// ---- DUTs/GreenMaster/IO/GreenMasterAI_Base.TcPOU
FUNCTION_BLOCK GreenMasterAI_Base
VAR_IN_OUT
	AIn: AnalogInputs;
END_VAR
VAR_INPUT
END_VAR
VAR_OUTPUT
	F_BT1_Error: BOOL;
	F_BT1: LREAL;
	T_BT2_Error: BOOL;
	T_BT2: LREAL;
	T_BT3_Error: BOOL;
	T_BT3: LREAL;
	H_BT1_Error: BOOL;
	H_BT1: LREAL;
	T_BT1_Error: BOOL;
	T_BT1: LREAL;
	BT1_Error: BOOL;
	BT1: LREAL;
	BT2_Error: BOOL;
	BT2: LREAL;
	F_BT2_Error: BOOL;
	F_BT2: LREAL;
END_VAR
VAR
END_VAR

END_FUNCTION_BLOCK

// ---- DUTs/GreenMaster/IO/GreenMasterAIU_Base.TcPOU
FUNCTION_BLOCK GreenMasterAIU_Base
VAR_INPUT
	EN: BOOL;
	T_BP2_Override: BOOL;
	T_BP2_OverrideValue: LREAL;
END_VAR
VAR_OUTPUT
	T_BF1_Error: BOOL;
	T_BF1: LREAL;
	F_BF1_Error: BOOL;
	F_BF1: LREAL;
	T_BP1_Error: BOOL;
	T_BP1: LREAL;
	F_BP1_Error: BOOL;
	F_BP1: LREAL;
	T_BP2_Error: BOOL;
	T_BP2: LREAL;
	F_BP2_Error: BOOL;
	F_BP2: LREAL;
	F_BP3_Error: BOOL;
	F_BP3: LREAL;
	T_CurrentPower: LREAL;
	F_CurrentPower: LREAL;
	T_CurrentSpeed: LREAL;
	F_CurrentSpeed: LREAL;
END_VAR
VAR
END_VAR

END_FUNCTION_BLOCK

// ---- DUTs/Parameters/IO/AnalogOutputParametersFB.TcPOU
FUNCTION_BLOCK AnalogOutputParametersFB
VAR_INPUT
END_VAR
VAR_OUTPUT
END_VAR
VAR
END_VAR

METHOD Update : BOOL
VAR_INPUT
	AO: REFERENCE TO GreenMasterAO_Base;
	Parameters: REFERENCE TO GreenMasterBaseParameters;
	AOut: AnalogOutputParameters;
END_VAR
VAR
	NotFire: BOOL;
END_VAR
NotFire := NOT Main.GreenMaster.FireAlarm();
AO.F_QN1 := ifc_lreal(Parameters.IO.AOutOverride.F_QN1_Override AND NotFire, Parameters.IO.AOutOverride.F_QN1_OverrideValue, AOut.F_QN1);
AO.T_GQ1 := ifc_lreal(Parameters.IO.AOutOverride.T_GQ1_Override AND NotFire, Parameters.IO.AOutOverride.T_GQ1_OverrideValue, AOut.T_GQ1);
AO.F_GQ1 := ifc_lreal(Parameters.IO.AOutOverride.F_GQ1_Override AND NotFire, Parameters.IO.AOutOverride.F_GQ1_OverrideValue, AOut.F_GQ1);
AO.C_QN1 := ifc_lreal(Parameters.IO.AOutOverride.C_QN1_Override AND NotFire, Parameters.IO.AOutOverride.C_QN1_OverrideValue, AOut.C_QN1);
AO.H_QN1 := ifc_lreal(Parameters.IO.AOutOverride.H_QN1_Override AND NotFire, Parameters.IO.AOutOverride.H_QN1_OverrideValue, AOut.H_QN1);
END_METHOD

END_FUNCTION_BLOCK

// ---- DUTs/GreenMaster/IO/GreenMasterAO_Base.TcPOU
FUNCTION_BLOCK GreenMasterAO_Base
VAR_IN_OUT
	AOut: AnalogOutputs;
END_VAR
VAR_INPUT
	F_QN1: LREAL;
	T_GQ1: LREAL;
	F_GQ1: LREAL;
	C_QN1: LREAL;
	H_QN1: LREAL;	
END_VAR
VAR_OUTPUT
END_VAR
VAR
END_VAR

METHOD SetOverrideF_GQ1 : BOOL
VAR_INPUT
	Override: BOOL;
	OverrideValue: LREAL;
	Parameters: REFERENCE TO GreenMasterBaseParameters;
END_VAR
END_METHOD

METHOD SetOverrideF_QN1 : BOOL
VAR_INPUT
	Override: BOOL;
	OverrideValue: LREAL;
	Parameters: REFERENCE TO GreenMasterBaseParameters;
END_VAR
END_METHOD

METHOD SetOverrideH_QN1 : BOOL
VAR_INPUT
	Override: BOOL;
	OverrideValue: LREAL;
	Parameters: REFERENCE TO GreenMasterBaseParameters;
END_VAR
END_METHOD

METHOD SetOverrideT_GQ1 : BOOL
VAR_INPUT
	Override: BOOL;
	OverrideValue: LREAL;
	Parameters: REFERENCE TO GreenMasterBaseParameters;
END_VAR
END_METHOD

END_FUNCTION_BLOCK

// ---- DUTs/Utilities/ifc_lreal.TcPOU
FUNCTION ifc_lreal : LREAL
VAR_INPUT
	Condition: BOOL;
	ValueTrue: LREAL;
	ValueFalse: LREAL;
END_VAR
VAR
END_VAR

IF Condition THEN
	ifc_lreal := ValueTrue;
ELSE
	ifc_lreal := ValueFalse;
END_IF

END_FUNCTION

// ---- DUTs/Utilities/BoolToErrorText.TcPOU
FUNCTION BoolToErrorText : STRING
VAR_INPUT
	Error: BOOL;
END_VAR
VAR
END_VAR

IF Error THEN
	BoolToErrorText := 'Error';
ELSE
	BoolToErrorText := 'OK';
END_IF

END_FUNCTION

// ---- DUTs/Parameters/Simulation/SimulationFB.TcPOU
FUNCTION_BLOCK SimulationFB
VAR_IN_OUT
	Parameters: GreenMasterBaseParameters;
END_VAR
VAR_INPUT
	Simulation: SimulationParameters;	
END_VAR
VAR_OUTPUT
END_VAR
VAR
END_VAR

Main.GreenMaster.Simulate(Parameters := Main.GreenMaster.GetParameters(),
	ParametersFB := Main.GreenMaster.GetParametersFB());

END_FUNCTION_BLOCK

// ---- DUTs/Parameters/SmokeControl/SmokeControlParametersBaseFB.TcPOU
FUNCTION_BLOCK SmokeControlParametersBaseFB
VAR_INPUT
END_VAR
VAR_OUTPUT
	NetLink: NetLinkParametersFB;
	DamperModules: SxDuoParametersFB;
END_VAR
VAR
END_VAR

END_FUNCTION_BLOCK

// ---- DUTs/Parameters/SmokeControl/NetLinkParametersFB.TcPOU
FUNCTION_BLOCK NetLinkParametersFB
VAR_INPUT
END_VAR
VAR_OUTPUT
END_VAR
VAR
END_VAR

METHOD Update : BOOL
VAR_INPUT
	Parameters: REFERENCE TO GreenMasterBaseParameters;
END_VAR
END_METHOD

END_FUNCTION_BLOCK

// ---- DUTs/Parameters/SmokeControl/SxDuoParametersFB.TcPOU
FUNCTION_BLOCK SxDuoParametersFB
VAR_INPUT
END_VAR
VAR_OUTPUT
	Unit01: SxDuoUnitFB;
	Unit02: SxDuoUnitFB;
	Unit03: SxDuoUnitFB;
	Unit04: SxDuoUnitFB;
	Unit05: SxDuoUnitFB;
	Unit06: SxDuoUnitFB;
	Unit07: SxDuoUnitFB;
	Unit08: SxDuoUnitFB;
	Unit09: SxDuoUnitFB;
	Unit10: SxDuoUnitFB;
	Unit11: SxDuoUnitFB;
	Unit12: SxDuoUnitFB;
	Unit13: SxDuoUnitFB;
	Unit14: SxDuoUnitFB;
	Unit15: SxDuoUnitFB;
END_VAR
VAR
END_VAR

END_FUNCTION_BLOCK

// ---- DUTs/Parameters/SmokeControl/SxDuoUnitFB.TcPOU
FUNCTION_BLOCK SxDuoUnitFB
VAR_INPUT
	Simulation: REFERENCE TO SimulationParameters;
END_VAR
VAR_OUTPUT
END_VAR
VAR
END_VAR

Simulation.ENO := Simulation.EN;

METHOD Update : BOOL
VAR_INPUT
	Parameters: REFERENCE TO GreenMasterBaseParameters;
	DamperModule: REFERENCE TO DamperModule;
	SxDuoUnit: REFERENCE TO SxDuoUnit;
END_VAR
SxDuoUnit.Error := DamperModule.Error;
SxDuoUnit.Fire := DamperModule.Fire;
SxDuoUnit.SxDuoStatus := DamperModule.SxDuoStatus;
DamperModule.SxDuoCommand := SxDuoUnit.SxDuoCommand;
SxDuoUnit.Text := DamperModule.Text;
SxDuoUnit.Text_CP1252 := DamperModule.Text_CP1252;
END_METHOD

END_FUNCTION_BLOCK

// ---- DUTs/Smoke Control/DamperModule.TcPOU
FUNCTION_BLOCK DamperModule
VAR_INPUT
	EN: BOOL;
	UnitID: BYTE;
	ModbusTCP: REFERENCE TO Modbus;
	Exercise: BOOL;
	ResetSmokeDetector: bool;
	SxDuoCommand: SxDuoCommand;
	{attribute 'TcEncoding':='UTF-8'}
	WriteText: STRING;
END_VAR
VAR_OUTPUT
	ENO: BOOL;
	Error: BOOL;
	Fire: BOOL;
	Exercising: BOOL;
	DamperError: BOOL;
	ServiceAlarm: BOOL;
	{attribute 'TcEncoding':='UTF-8'}
	Text: STRING;
	Text_CP1252: STRING;
	SxDuoStatus: SxDuoStatus;
END_VAR
VAR
	ModbusReadBits3: ModbusReadBits;
	ModbusWriteBits3: ModbusWriteBits;
	ModbusReadWordArray_0: ModbusReadWordArray;
END_VAR
VAR // added by the converter: edge detectors and wires of the graphical bodies
    _s1 : SxDuoStatus;
    _w1, _w2 : ANY;
END_VAR


// PAGE
ModbusWriteBits3(
    EN := EN,
    Modbus := ModbusTCP,
    UnitID := UnitID,
    Register := 44,
    b1 := ???,
    b2 := _w1,
    b4 := _w2); // ModbusWriteBits
ModbusReadBits3(EN := EN, Modbus := ModbusTCP, UnitID := UnitID, Register := 32); // ModbusReadBits
Error := ModbusReadBits3.Error;
Fire := ModbusReadBits3.b1;
_w2 := Exercise OR ???;
Exercising := ModbusReadBits3.b4;
DamperError := ModbusReadBits3.b6;
// compose _s1 : SxDuoStatus
_s1.FireAlarm := ModbusReadBits3.b1;
_s1.Damper1Alarm := ModbusReadBits3.b3;
_s1.Exercising := ModbusReadBits3.b4;
_s1.Damper2Alarm := ModbusReadBits3.b5;
_s1.Damper1Open := ModbusReadBits3.b9;
_s1.Damper1Closed := ModbusReadBits3.b8;
_s1.Damper2Open := ModbusReadBits3.b11;
_s1.Damper2Closed := ModbusReadBits3.b10;
_s1.ServiceAlarm := ModbusReadBits3.b14;
SxDuoStatus := _s1;
_w1 := ResetSmokeDetector OR ???;
ServiceAlarm := ModbusReadBits3.b14;
ModbusReadWordArray_0(
    EN := EN,
    Modbus := ModbusTCP,
    UnitID := UnitID,
    RegisterType := ModbusRegisterType.HoldingRegister,
    Register := 16#8000 + 16#110,
    ParameterCount := 16,
    UpdateInterval := LTIME#1m,
    WriteText := WriteText); // ModbusReadWordArray
Text := ModbusReadWordArray_0.Text;
Text_CP1252 := ModbusReadWordArray_0.Text_CP1252;

METHOD StartWrite : BOOL
VAR_INPUT
END_VAR
ModbusWriteBits3.EN := TRUE;
END_METHOD

END_FUNCTION_BLOCK

// ---- DUTs/ModbusTCP/ModbusTCP.TcPOU
FUNCTION_BLOCK ModbusTCP EXTENDS Modbus
VAR_INPUT
	EN: BOOL;
	{attribute 'TcEncoding':='UTF-8'}
	IP: STRING;
	Port: UINT := 502;
END_VAR
VAR_OUTPUT
	ENO: BOOL;
	Error: BOOL;
END_VAR
VAR
	ModbusMaster: FB_MBReadRegs;
	ModbusMasterWrite: FB_MBWriteRegs;
	{attribute 'TcEncoding':='UTF-8'}
	stMbErrId: STRING;
	aRegisterArray1: ARRAY [1..125] OF WORD;
	aRegisterCoil: ARRAY [1..250] OF BYTE;
	WaitModbusBusy: TON;
	cbRead: INT;
	Param: REFERENCE TO ModbusIo;
	State: INT;
	ReplyTON: LTON;
	LastReadCount: LINT;
END_VAR
VAR PERSISTENT
	tTimeBetweenReads: TIME := T#100MS;
END_VAR

SUPER^();
ENO := EN;
ReplyTON(IN := ReadCount = LastReadCount, PT := LTIME#20S, Q => Error);
LastReadCount := ReadCount;
WaitModbusBusy();
CASE State OF
	0:
		IF EN THEN		
			CurrentIoIndex := 0;
			IF IO[CurrentIoIndex] <> 0 THEN
				State := 5;
			END_IF	
		END_IF
	5:	(* Wait between reads *)
		WaitModbusBusy(IN := TRUE, PT := tTimeBetweenReads, Q=> , ET=> );	
		IF WaitModbusBusy.Q = TRUE THEN
			IF TIME_TO_LTIME(NowDT() - IO[CurrentIoIndex]^.LastUpdate) > IO[CurrentIoIndex]^.UpdateInterval THEN	
				IO[CurrentIoIndex]^.SetLastUpdate(NowDT());			
				IF NOT IO[CurrentIoIndex]^.Write THEN
					State := 10;
				ELSE
					State := 110;			
				END_IF
			ELSE
				State := 30;
			END_IF
			WaitModbusBusy(IN := FALSE);
		END_IF		
	
	10:
		Param REF= IO[CurrentIoIndex]^; 
		IF NOT Param.EN OR Param.UnitID = 0 THEN
			Param.ValueWord := 0;
			Param.ErrorOUT := FALSE;
			State := 30;
		ELSE
			ModbusMaster(
			sIPAddr:= IP, 
			nTCPPort:= 502, 
			nUnitID:= Param.UnitID, 
			nQuantity:= Param.ParameterCount, 
			nMBAddr:= Param.Register, 
			cbLength:= 2 * Param.ParameterCount, 
			pDestAddr:= ADR(aRegisterArray1), 
			bExecute:= TRUE, 
			tTimeout:= T#1000MS);
			IF  ModbusMaster.bBUSY THEN
				State := State + 10;
			END_IF
		END_IF
	20:
		ModbusMaster();
		IF ModbusMaster.bError THEN
			stMbErrId := concat('Error ', UDINT_TO_STRING(ModbusMaster.nErrId));
			ModbusMaster(bExecute := FALSE);
			Param.ValueWord := 0;
			Param.ErrorOUT := TRUE;
			ErrorCount := ErrorCount + 1;
			ModbusMaster.bExecute:= FALSE;
			State := 30;
		ELSIF NOT ModbusMaster.bBUSY THEN
			ModbusMaster(bExecute := FALSE);
			Param.ValueWord := aRegisterArray1[1];
			Param.ValueWordArray := aRegisterArray1;
			Param.ErrorOUT := FALSE;
			ReadCount := ReadCount + 1;
			ModbusMaster(bExecute:= FALSE);
			State := 30;
		END_IF
	30:
		CurrentIoIndex := CurrentIoIndex + 1;
		IF CurrentIoIndex >= IO_COUNT THEN
			CurrentIoIndex := 0;
		END_IF
		IF IO[CurrentIoIndex] <> 0 THEN
			State := 5;
		ELSE				
			State := 0;
		END_IF
	110:
		Param REF= IO[CurrentIoIndex]^; 
		IF NOT Param.EN OR Param.UnitID = 0 THEN
			Param.ValueWord := 0;
			Param.ErrorOUT := FALSE;
			State := 30;
		ELSE
			aRegisterArray1[1] := Param.ValueWord;
			ModbusMasterWrite(
			sIPAddr:= IP, 
			nTCPPort:= 502, 
			nUnitID:= Param.UnitID, 
			nQuantity:= Param.ParameterCount, 
			nMBAddr:= Param.Register, 
			cbLength:= 2 * Param.ParameterCount, 
			pSrcAddr:= ADR(aRegisterArray1), 
			bExecute:= TRUE, 
			tTimeout:= T#1000MS);
			IF  ModbusMasterWrite.bBUSY THEN
				State := State + 10;
			END_IF
		END_IF
	120:
		ModbusMasterWrite();
		IF ModbusMasterWrite.bError THEN
			stMbErrId := concat('Error ', UDINT_TO_STRING(ModbusMaster.nErrId));
			ModbusMasterWrite(bExecute := FALSE);
			Param.ValueWord := 0;
			Param.ErrorOUT := TRUE;
			ErrorCount := ErrorCount + 1;
			ModbusMasterWrite.bExecute:= FALSE;
			State := 30;
		ELSIF NOT ModbusMasterWrite.bBUSY THEN
			ModbusMasterWrite(bExecute := FALSE);
			Param.ValueWord := aRegisterArray1[1];
			Param.ValueWordArray := aRegisterArray1;
			Param.ErrorOUT := FALSE;
			ReadCount := ReadCount + 1;
			ModbusMasterWrite(bExecute:= FALSE);
			State := 30;
		END_IF
		Param.EN := FALSE;
		Param.Write := FALSE;
END_CASE

END_FUNCTION_BLOCK

// ---- DUTs/ModbusRTU/Modbus.TcPOU
FUNCTION_BLOCK Modbus
VAR_INPUT
END_VAR
VAR_OUTPUT
	ReadCount: LINT;
	ErrorCount: LINT;
END_VAR
VAR CONSTANT
	IO_COUNT: INT := 100;
END_VAR
VAR
	Self: REFERENCE TO Modbus;
	IO: ARRAY [0..IO_COUNT - 1] OF POINTER TO ModbusIo;
	IOIndex: INT;
	CurrentIoIndex: INT;
END_VAR

Self REF= THIS^;

METHOD AddIO : BOOL
VAR_INPUT
	Self: pointer TO ModbusIO {flag write};
END_VAR
IF IOIndex < IO_COUNT THEN
	IO[IOIndex] := Self;
	IOIndex := IOIndex + 1;
END_IF
END_METHOD

END_FUNCTION_BLOCK

// ---- DUTs/ModbusRTU/ModbusIo.TcPOU
FUNCTION_BLOCK ModbusIo
VAR_INPUT
	EN: BOOL := TRUE;
	Modbus: REFERENCE TO Modbus;
	UnitID: BYTE;
	RegisterType: ModbusRegisterType;
	Register: WORD;
	Write: BOOL := FALSE;
	ParameterCount: WORD := 1;
	UpdateInterval: LTIME := LTIME#2S;
END_VAR
VAR_OUTPUT
	ENO: BOOL;
	Error: BOOL;
	LastUpdate: DT;
END_VAR
VAR_IN_OUT
END_VAR
VAR
	Registered: BOOL;
	ErrorCount: INT;
END_VAR
VAR PERSISTENT
END_VAR

IF EN AND __ISVALIDREF(Modbus) THEN
	IF NOT Registered THEN
		Modbus.AddIO(THIS);
		Registered := TRUE;	
	END_IF
END_IF
ENO := EN and not Error;

PROPERTY ErrorOut : BOOL
GET
ErrorOut := Error;
END_GET
SET
Error := ErrorOut;
END_SET
END_PROPERTY

METHOD GetErrorCount : INT
VAR_INPUT
END_VAR
GetErrorCount := ErrorCount;
END_METHOD

METHOD IncErrorCount : BOOL
VAR_INPUT
END_VAR
IF ErrorCount < 10 THEN
	ErrorCount := ErrorCount + 1;
END_IF
END_METHOD

METHOD ResetErrorCount : BOOL
VAR_INPUT
END_VAR
ErrorCount := 0;
END_METHOD

METHOD SetLastUpdate : BOOL
VAR_INPUT
	CurrentTime: DT;
END_VAR
LastUpdate := CurrentTime;
END_METHOD

PROPERTY ValueBoolOut : BOOL
GET
END_GET
SET
END_SET
END_PROPERTY

PROPERTY ValueWord : WORD
GET
END_GET
SET
END_SET
END_PROPERTY

PROPERTY ValueWordArray : ARRAY [1..125] OF WORD
GET
END_GET
SET
END_SET
END_PROPERTY

END_FUNCTION_BLOCK

// ---- DUTs/ModbusRTU/ModbusReadBits.TcPOU
FUNCTION_BLOCK ModbusReadBits EXTENDS ModbusIo
VAR_INPUT
END_VAR
VAR_OUTPUT
	b0: BOOL;
	b1: BOOL;
	b2: BOOL;
	b3: BOOL;
	b4: BOOL;
	b5: BOOL;
	b6: BOOL;
	b7: BOOL;
	b8: BOOL;
	b9: BOOL;
	b10: BOOL;
	b11: BOOL;
	b12: BOOL;
	b13: BOOL;
	b14: BOOL;
	b15: BOOL;
END_VAR
VAR
END_VAR

SUPER^();

PROPERTY ValueWord : WORD
GET
ValueWord := 0;
IF b0 THEN
	ValueWord := ValueWord OR 16#0001;
END_IF
IF b1 THEN
	ValueWord := ValueWord OR 16#0002;
END_IF
IF b2 THEN
	ValueWord := ValueWord OR 16#0004;
END_IF
IF b3 THEN
	ValueWord := ValueWord OR 16#0008;
END_IF
IF b4 THEN
	ValueWord := ValueWord OR 16#0010;
END_IF
IF b5 THEN
	ValueWord := ValueWord OR 16#0020;
END_IF
IF b6 THEN
	ValueWord := ValueWord OR 16#0040;
END_IF
IF b7 THEN
	ValueWord := ValueWord OR 16#0080;
END_IF
IF b8 THEN
	ValueWord := ValueWord OR 16#0100;
END_IF
IF b9 THEN
	ValueWord := ValueWord OR 16#0200;
END_IF
IF b10 THEN
	ValueWord := ValueWord OR 16#0400;
END_IF
IF b11 THEN
	ValueWord := ValueWord OR 16#0800;
END_IF
IF b12 THEN
	ValueWord := ValueWord OR 16#1000;
END_IF
IF b13 THEN
	ValueWord := ValueWord OR 16#2000;
END_IF
IF b14 THEN
	ValueWord := ValueWord OR 16#4000;
END_IF
IF b15 THEN
	ValueWord := ValueWord OR 16#8000;
END_IF
END_GET
SET
b0 := (ValueWord AND 16#0001) <> 0;
b1 := (ValueWord AND 16#0002) <> 0;
b2 := (ValueWord AND 16#0004) <> 0;
b3 := (ValueWord AND 16#0008) <> 0;
b4 := (ValueWord AND 16#0010) <> 0;
b5 := (ValueWord AND 16#0020) <> 0;
b6 := (ValueWord AND 16#0040) <> 0;
b7 := (ValueWord AND 16#0080) <> 0;
b8 := (ValueWord AND 16#0100) <> 0;
b9 := (ValueWord AND 16#0200) <> 0;
b10 := (ValueWord AND 16#0400) <> 0;
b11 := (ValueWord AND 16#0800) <> 0;
b12 := (ValueWord AND 16#1000) <> 0;
b13 := (ValueWord AND 16#2000) <> 0;
b14 := (ValueWord AND 16#4000) <> 0;
b15 := (ValueWord AND 16#8000) <> 0;
END_SET
END_PROPERTY

END_FUNCTION_BLOCK

// ---- DUTs/ModbusRTU/ModbusWriteBits.TcPOU
FUNCTION_BLOCK ModbusWriteBits EXTENDS ModbusIo
VAR_INPUT
	b0: BOOL;
	b1: BOOL;
	b2: BOOL;
	b3: BOOL;
	b4: BOOL;
	b5: BOOL;
	b6: BOOL;
	b7: BOOL;
	b8: BOOL;
	b9: BOOL;
	b10: BOOL;
	b11: BOOL;
	b12: BOOL;
	b13: BOOL;
	b14: BOOL;
	b15: BOOL;
END_VAR
VAR_OUTPUT
END_VAR
VAR
	Pre_b0: BOOL;
	Pre_b1: BOOL;
	Pre_b2: BOOL;
	Pre_b3: BOOL;
	Pre_b4: BOOL;
	Pre_b5: BOOL;
	Pre_b6: BOOL;
	Pre_b7: BOOL;
	Pre_b8: BOOL;
	Pre_b9: BOOL;
	Pre_b10: BOOL;
	Pre_b11: BOOL;
	Pre_b12: BOOL;
	Pre_b13: BOOL;
	Pre_b14: BOOL;
	Pre_b15: BOOL;
END_VAR

SUPER^();
IF 
	(b0 <> Pre_b0) OR
	(b1 <> Pre_b1) OR
	(b2 <> Pre_b2) OR
	(b3 <> Pre_b3) OR
	(b4 <> Pre_b4) OR
	(b5 <> Pre_b5) OR
	(b6 <> Pre_b6) OR
	(b7 <> Pre_b7) OR
	(b8 <> Pre_b8) OR
	(b9 <> Pre_b9) OR
	(b10 <> Pre_b10) OR
	(b11 <> Pre_b11) OR
	(b12 <> Pre_b12) OR
	(b13 <> Pre_b13) OR
	(b14 <> Pre_b14) OR
	(b15 <> Pre_b15) THEN
	Pre_b0 := b0;
	Pre_b1 := b1;
	Pre_b2 := b2;
	Pre_b3 := b3;
	Pre_b4 := b4;
	Pre_b5 := b5;
	Pre_b6 := b6;
	Pre_b7 := b7;
	Pre_b8 := b8;
	Pre_b9 := b9;
	Pre_b10 := b10;
	Pre_b11 := b11;
	Pre_b12 := b12;
	Pre_b13 := b13;
	Pre_b14 := b14;
	Pre_b15 := b15;
	Write := TRUE;
END_IF

PROPERTY ValueWord : WORD
GET
ValueWord := 0;
IF b0 THEN
	ValueWord := ValueWord OR 16#0001;
END_IF
IF b1 THEN
	ValueWord := ValueWord OR 16#0002;
END_IF
IF b2 THEN
	ValueWord := ValueWord OR 16#0004;
END_IF
IF b3 THEN
	ValueWord := ValueWord OR 16#0008;
END_IF
IF b4 THEN
	ValueWord := ValueWord OR 16#0010;
END_IF
IF b5 THEN
	ValueWord := ValueWord OR 16#0020;
END_IF
IF b6 THEN
	ValueWord := ValueWord OR 16#0040;
END_IF
IF b7 THEN
	ValueWord := ValueWord OR 16#0080;
END_IF
IF b8 THEN
	ValueWord := ValueWord OR 16#0100;
END_IF
IF b9 THEN
	ValueWord := ValueWord OR 16#0200;
END_IF
IF b10 THEN
	ValueWord := ValueWord OR 16#0400;
END_IF
IF b11 THEN
	ValueWord := ValueWord OR 16#0800;
END_IF
IF b12 THEN
	ValueWord := ValueWord OR 16#1000;
END_IF
IF b13 THEN
	ValueWord := ValueWord OR 16#2000;
END_IF
IF b14 THEN
	ValueWord := ValueWord OR 16#4000;
END_IF
IF b15 THEN
	ValueWord := ValueWord OR 16#8000;
END_IF
END_GET
SET
b0 := (ValueWord AND 16#0001) <> 0;
b1 := (ValueWord AND 16#0002) <> 0;
b2 := (ValueWord AND 16#0004) <> 0;
b3 := (ValueWord AND 16#0008) <> 0;
b4 := (ValueWord AND 16#0010) <> 0;
b5 := (ValueWord AND 16#0020) <> 0;
b6 := (ValueWord AND 16#0040) <> 0;
b7 := (ValueWord AND 16#0080) <> 0;
b8 := (ValueWord AND 16#0100) <> 0;
b9 := (ValueWord AND 16#0200) <> 0;
b10 := (ValueWord AND 16#0400) <> 0;
b11 := (ValueWord AND 16#0800) <> 0;
b12 := (ValueWord AND 16#1000) <> 0;
b13 := (ValueWord AND 16#2000) <> 0;
b14 := (ValueWord AND 16#4000) <> 0;
b15 := (ValueWord AND 16#8000) <> 0;
END_SET
END_PROPERTY

END_FUNCTION_BLOCK

// ---- DUTs/ModbusRTU/ModbusReadWordArray.TcPOU
FUNCTION_BLOCK ModbusReadWordArray EXTENDS ModbusIo
VAR_INPUT
	{attribute 'TcEncoding':='UTF-8'}
	WriteText: STRING;
END_VAR
VAR_OUTPUT
	Value: ARRAY [1..125] OF WORD;
	{attribute 'TcEncoding':='UTF-8'}
	Text: STRING;
	Text_CP1252: STRING;
END_VAR
VAR
END_VAR
VAR PERSISTENT
END_VAR

SUPER^();
Text := GetText();
Text_CP1252 := GetText_CP1252();
SetText(WriteText);

{attribute 'TcEncoding':='UTF-8'}
METHOD GetText : string
VAR_INPUT
END_VAR
VAR
	//{attribute 'TcEncoding':='UTF-8'}
	Str: STRING;
	arr: ARRAY [1..125] OF WORD;
	p: POINTER TO ARRAY [0..MAX_STRING_LENGTH] OF BYTE;
	n: INT;
	{attribute 'TcEncoding':='UTF-8'}
	Utf8: STRING;
END_VAR
arr := Value;
FOR n := 1 TO 125 DO
	arr[n] := SHR(arr[n] AND 16#FF00, 8) + SHL(arr[n] AND 16#00FF, 8);
END_FOR
p := ADR(arr);
Str := BYTEARR_TO_MAXSTRING(p^);
STRING_TO_UTF8(ADR(Utf8), ADR(Str), SIZEOF(Utf8));
GetText := Utf8;
END_METHOD

METHOD GetText_CP1252 : STRING
VAR_INPUT
END_VAR
VAR
	Str: STRING;
	arr: ARRAY [1..125] OF WORD;
	p: POINTER TO ARRAY [0..MAX_STRING_LENGTH] OF BYTE;
	n: INT;
END_VAR
arr := Value;
FOR n := 1 TO 125 DO
	arr[n] := SHR(arr[n] AND 16#FF00, 8) + SHL(arr[n] AND 16#00FF, 8);
END_FOR
p := ADR(arr);
Str := BYTEARR_TO_MAXSTRING(p^);
GetText_CP1252 := Str;
END_METHOD

METHOD SetText : BOOL
VAR_INPUT
	{attribute 'TcEncoding':='UTF-8'}
	NewText: STRING;
END_VAR
VAR
	Str: STRING;
	TempValue, TestValue: ARRAY [1..125] OF WORD;
	bArr: ARRAY [0..MAX_STRING_LENGTH] OF BYTE;
	n: INT;
	{attribute 'TcEncoding':='UTF-8'}
	nDstLen: UDINT;
	byte0, byte1: BYTE;
	numWords: INT;
END_VAR
(*
IF UTF8_TO_STRING(ADR(Str), ADR(NewText), SIZEOF(Str), nDstLen => nDstLen) THEN	
	bArr := MAXSTRING_TO_BYTEARR(Str);
	bArr[nDstLen] := 0;
	nDstLen := nDstLen + 1;
	TempValue := Value;
	numWords := UDINT_TO_INT(nDstLen / 2);
	IF (nDstLen AND 1) <> 0 THEN
		numWords := numWords + 1;
	END_IF
	FOR n := 0 TO numWords - 1 DO
		IF (n * 2 + 1) < UDINT_TO_INT(nDstLen) THEN
			byte0 := bArr[n * 2 + 1];
		ELSE
			byte0 := 0;		
		END_IF
		byte1 := bArr[n * 2];
		TempValue[n + 1] := SHL(BYTE_TO_WORD(byte0), 8) + byte1;
	END_FOR
	IF NOT AnyEqual(TempValue, Value) THEN
		TestValue := TempValue;
		//Value := TempValue;
		//Write := TRUE;
	END_IF
END_IF
*)
END_METHOD

PROPERTY TextValue : STRING
GET
TextValue := GetText();
END_GET
SET
SetText(TextValue);
END_SET
END_PROPERTY

PROPERTY ValueWordArray : array [1..125] of WORD
GET
ValueWordArray := Value;
END_GET
SET
Value := ValueWordArray;
END_SET
END_PROPERTY

END_FUNCTION_BLOCK

// ---- DUTs/Utilities/WriteBoolIf.TcPOU
FUNCTION_BLOCK WriteBoolIf
VAR_IN_OUT
	Out: BOOL;
END_VAR
VAR_INPUT
	EN: BOOL := TRUE;
	In: BOOL;
END_VAR
VAR_OUTPUT
	ENO: BOOL;
END_VAR
VAR
END_VAR

ENO := EN;
IF EN THEN
	Out := In;
END_IF

END_FUNCTION_BLOCK

// ---- DUTs/Exercise/ExerciseF_P1.TcPOU
FUNCTION_BLOCK ExerciseF_P1
VAR_IN_OUT
	Parameters: GreenMasterBaseParameters;
END_VAR
VAR_INPUT
	EN: BOOL := TRUE;
	ForceExercise: BOOL;
END_VAR
VAR_OUTPUT
	Exercising: BOOL;
END_VAR
VAR
	ExerciseTimer: Timer;
	LocalTime: FB_LocalSystemTime;
	Elapsed: LINT;
	CurrentState: INT;
	StateTimer: TImer;
	DetectedDamperError: BOOL;
	FirstTime: BOOL := TRUE;
END_VAR

LocalTime(bEnable := TRUE);
ExerciseTimer(EN := EN);
Elapsed := ExerciseTimer.ElapsedTime();

StateTimer();
IF EN THEN
	CASE CurrentState OF
		0:
			IF EN AND LocalTime.bValid THEN
				IF ((Parameters.System.Exercise.CirculationPumps.Interval > 0) AND ((ExerciseTimer.ElapsedTime() > (Parameters.System.Exercise.CirculationPumps.Interval * 3600 * 1000)) OR FirstTime) AND 
					(
						(WORD_TO_INT(LocalTime.systemTime.wHour) = Parameters.System.Exercise.CirculationPumps.Hour) AND (WORD_TO_INT(LocalTime.systemTime.wMinute) = Parameters.System.Exercise.CirculationPumps.Minute)
					)) OR ForceExercise THEN
					FirstTime := FALSE;
					ForceExercise := FALSE;
					Exercising := TRUE;
					StateTimer.Restart();
					CurrentState := 1;
					Main.EventLog.LogEvent(EventTypes.Information, 'Exercising P1');
				END_IF			
			END_IF
		1:
			IF StateTimer.ElapsedTime() > 60 * 1000 THEN
				Exercising := FALSE;
				CurrentState := 0;
			END_IF
	END_CASE
END_IF

END_FUNCTION_BLOCK

// ---- DUTs/Events/EventLog.TcPOU
FUNCTION_BLOCK EventLog
VAR_IN_OUT
	EventLogData: EventLogData;	
END_VAR
VAR_INPUT
END_VAR
VAR_OUTPUT
END_VAR
VAR
	StartupDone: BOOL;
	EventLogDataRef: reference to EventLogData;	
	IncludeJSON: BOOL;
	sJSON: STRING(2000);
	fbJsonDataType: FB_JsonReadWriteDataType;
END_VAR

IF NOT StartupDone THEN
	EventLogDataRef REF= EventLogData;
	StartupDone := TRUE;
END_IF

METHOD LogEvent : BOOL
VAR_INPUT
	Kind: EventTypes := EventTypes.Information;
	Message: STRING;
END_VAR
VAR
	TempHead, TempTail: INT;
	n: uint;
END_VAR
IF __ISVALIDREF(EventLogDataRef) THEN
	TempTail := EventLogDataRef.Tail + 1;
	IF TempTail > Globals.EventsHigh THEN
		TempTail := Globals.EventsLow;
	END_IF
	
	IF TempTail = EventLogDataRef.Head THEN
		TempHead := EventLogDataRef.Head + 1;
		IF TempHead > Globals.EventsHigh THEN
			TempHead := Globals.EventsLow;
		END_IF
		EventLogDataRef.Head := TempHead;
	END_IF
	
	EventLogDataRef.Events[EventLogDataRef.Tail].Kind := Kind;
	EventLogDataRef.Events[EventLogDataRef.Tail].TimeStamp := NowDT();
	EventLogDataRef.Events[EventLogDataRef.Tail].Message := Message;
	n:= INT_TO_UINT(Len(sJSON));
	n :=  SIZEOF(EventLogDataRef.Events[EventLogDataRef.Tail].JSON);
	IF IncludeJSON AND (INT_TO_UINT(Len(sJSON)) < SIZEOF(Globals.EventLogStrings[EventLogDataRef.Tail])) THEN
		Globals.EventLogStrings[EventLogDataRef.Tail] := sJSON;
		EventLogDataRef.Events[EventLogDataRef.Tail].JSON := TRUE;
	ELSE
		EventLogDataRef.Events[EventLogDataRef.Tail].JSON := FALSE;
	END_IF
	
	EventLogDataRef.Tail := TempTail;
END_IF
END_METHOD

METHOD LogEventJSON : BOOL
VAR_INPUT
	Kind: EventTypes := EventTypes.Information;
	Message: STRING;
	VarType: STRING;
	VarSize: DWORD;
	VarAdr: POINTER TO DWORD;
END_VAR
VAR
	nLen: UDINT;
END_VAR
sJSON := '';
nLen := fbJsonDataType.CopyJsonStringFromSymbol(VarType, VarSize, VarAdr, sJSON,SIZEOF(sJSON));
IF nLen > 0 THEN
	IF sJSON[0] <> F_ToASC('{') THEN
		sJSON := concat(concat('{ "Value": ', sJSON), ' }');
	END_IF
END_IF
IncludeJSON := nLen > 0;
LogEvent(Kind := Kind, Message := Message);
IncludeJSON := FALSE;
END_METHOD

END_FUNCTION_BLOCK

// ---- DUTs/Utilities/DeviationMonitor.TcPOU
FUNCTION_BLOCK DeviationMonitor
VAR_INPUT
	EN: BOOL := TRUE;
	Value: LREAL;
	TargetValue: LREAL := 100;
	DiffAllowed: LREAL := 5;
	Mode: DeviationMonitorMode := DeviationMonitorMode.Diff;
	Hysteresis: LREAL := 2;
	OnDelay: LTIME := LTIME#10S;
	OffDelay: LTIME := LTIME#5S;
END_VAR
VAR_OUTPUT
	ENO: BOOL;
	Error: BOOL;
END_VAR
VAR
	TempError: BOOL;
	Hyst: Hysteresis;
	UseValue: LREAL;
	UseTargetValue: LREAL;
	OnTON: TON;
	OffTOF: TOF;
END_VAR

UseValue  := Value;
UseTargetValue := TargetValue;
IF Mode = DeviationMonitorMode.Diff THEN
	UseValue := ABS(UseValue - TargetValue);	
	UseTargetValue := DiffAllowed;
END_IF
Hyst(Value := UseValue, LimitValue := UseTargetValue, Offset := Hysteresis);
IF EN and (Main.GreenMaster.GetParameters().System.Operation.State = SystemStates.Run) THEN
	IF (Mode = DeviationMonitorMode.Above) OR (Mode = DeviationMonitorMode.Diff) THEN
		TempError := Hyst.Above;
	ELSIF Mode = DeviationMonitorMode.Below THEN
		TempError := Hyst.Below;	
	END_IF
	IF Main.GreenMaster.GetParameters().System.Operation.State <> SystemStates.Run THEN
		TempError := False;
	END_IF
	OnTON(IN := TempError, PT := TO_TIME(OnDelay));
	OffTOF(IN := NOT TempError, PT := TO_TIME(OnDelay));
	IF OnTON.Q THEN
		Error := TRUE;
	END_IF
	IF OffTOF.Q THEN
		Error := FALSE;
	END_IF
ELSE
	Error := FALSE;
END_IF
ENO := EN;

END_FUNCTION_BLOCK

// ---- DUTs/GreenMaster/IO/GreenMasterSmokeControl_Base.TcPOU
FUNCTION_BLOCK GreenMasterSmokeControl_Base
VAR_IN_OUT
	Parameters: GreenMasterBaseParameters;	
	ParametersSC: SmokeControlParametersBase;
END_VAR
VAR_INPUT
	EN: BOOL;
END_VAR
VAR_OUTPUT
	FireAlarm: BOOL;
END_VAR
VAR
END_VAR

END_FUNCTION_BLOCK

// ---- DUTs/Exercise/ExerciseF_QM2.TcPOU
FUNCTION_BLOCK ExerciseF_QM2
VAR_IN_OUT
	Parameters: GreenMasterBaseParameters;
END_VAR
VAR_INPUT
	EN: BOOL := TRUE;
	ForceExercise: BOOL;
END_VAR
VAR_OUTPUT
	Exercising: BOOL;
END_VAR
VAR
	ExerciseTimer: Timer;
	LocalTime: FB_LocalSystemTime;
	Elapsed: LINT;
	CurrentState: INT;
	StateTimer: TImer;
	DetectedDamperError: BOOL;
	FirstTime: BOOL := TRUE;
END_VAR

LocalTime(bEnable := TRUE);
ExerciseTimer(EN := EN);
Elapsed := ExerciseTimer.ElapsedTime();

StateTimer();
IF EN THEN
	CASE CurrentState OF
		0:
			IF EN AND LocalTime.bValid THEN
				IF ((Parameters.System.Exercise.FireBypassDamper.Interval > 0) AND ((ExerciseTimer.ElapsedTime() > (Parameters.System.Exercise.FireBypassDamper.Interval * 3600 * 1000)) OR FirstTime) AND 
					(
						(WORD_TO_INT(LocalTime.systemTime.wHour) = Parameters.System.Exercise.FireBypassDamper.Hour) AND (WORD_TO_INT(LocalTime.systemTime.wMinute) = Parameters.System.Exercise.FireBypassDamper.Minute)
					)) OR ForceExercise THEN
					FirstTime := FALSE;
					ForceExercise := FALSE;
					Exercising := TRUE;
					StateTimer.Restart();
					CurrentState := 1;
					Main.EventLog.LogEvent(EventTypes.Information, 'Exercising F_QM2');
				END_IF			
			END_IF
		1:
			IF StateTimer.ElapsedTime() > 10 * 1000 THEN
				ExerciseTimer.Restart();
				Parameters.IO.DOut.F_QM2 := FALSE;
				CurrentState := 2;
			END_IF
		2:
			IF StateTimer.ElapsedTime() > 30 * 1000 THEN
				CurrentState := 3;
			END_IF
		3:
			IF (StateTimer.ElapsedTime() > 180 * 1000) or Parameters.IO.DIn.F_QM2_Closed THEN
				Parameters.IO.DOut.F_QM2 := TRUE;
				Exercising := FALSE;
				CurrentState := 0;
			END_IF
	END_CASE
END_IF

END_FUNCTION_BLOCK

// ---- DUTs/Alarms/AlarmMonitor.TcPOU
FUNCTION_BLOCK AlarmMonitor
VAR_IN_OUT
	AlarmLog: AlarmLog;
	Parameters: GreenMasterBaseParameters;
END_VAR
VAR_INPUT
	EN: BOOL;
	Reset: BOOL;
END_VAR
VAR_OUTPUT
	ENO: BOOL;
	AlarmA: BOOL;
	AlarmB: BOOL;
	AlarmC: BOOL;
	AlarmD: BOOL;
END_VAR
VAR
	AlarmSignals1: REFERENCE TO AlarmSignals;
	StartupDone: BOOL;
	AlarmLogRef: REFERENCE TO AlarmLog;
	NoAlarms, Current: AlarmEvent;
	n: UINT;
	aTON: ARRAY [0..19] OF TON;
	bTON: ARRAY [0..11] OF TON;
	cTON: ARRAY [0..3] OF TON;
	CurrentDT, LastDT: DATE_AND_TIME;
	IncludeJSON: BOOL;
	sJSON: STRING(2000);
	fbJsonDataType: FB_JsonReadWriteDataType;
	StartTime: Timer;
	Latched, Last: AlarmEvent;
	LastIoStatus: IoStatus;
	
	AlarmCount: UINT := SIZEOF(AlarmSignals);
	LatchedStatusP: POINTER TO ARRAY [0..SIZEOF(AlarmSignals) - 1] OF BOOL;
	LatchedSignalP: POINTER TO ARRAY [0..SIZEOF(AlarmSignals) - 1] OF BOOL;
	StatusP: POINTER TO ARRAY [0..SIZEOF(AlarmSignals) - 1] OF BOOL;
	AutoResetP: POINTER TO ARRAY [0..SIZEOF(AlarmSignals) - 1] OF BOOL;
	EnabledP: POINTER TO ARRAY [0..SIZEOF(AlarmSignals) - 1] OF BOOL;
	CurrentP: POINTER TO ARRAY [0..SIZEOF(AlarmSignals) - 1] OF BOOL;
	PolarityP: POINTER TO ARRAY [0..SIZEOF(AlarmSignals) - 1] OF BOOL;
	DelayP: POINTER TO ARRAY [0..SIZEOF(AlarmSignals) - 1] OF TIME;
	TONs: ARRAY [0..SIZEOF(AlarmSignals) - 1] OF TON;
	StartupDelay: TON;
END_VAR

IF NOT StartupDone THEN
	AlarmLogRef REF= AlarmLog;
	StartupDone := TRUE;
	AlarmSignals1 REF= Parameters.Alarm.Status;
END_IF
StartupDelay(IN := TRUE, PT := T#5S);
IF StartupDelay.Q THEN
	LatchedStatusP := ADR(Latched.Status);
	DelayP := ADR(Parameters.Alarm.Delay);
	StatusP := ADR(Parameters.Alarm.Status);
	PolarityP := ADR(Parameters.Alarm.Polarity);
	CurrentP := ADR(Current.Signals);
	EnabledP := ADR(Parameters.Alarm.Enabled);
	FOR N := 0 TO AlarmCount - 1 DO
		LatchedStatusP^[n] := (StatusP^[n] <> PolarityP^[n]) AND EnabledP^[n];		
		TONs[n](IN := LatchedStatusP^[n], PT := DelayP^[n], Q => CurrentP^[n]);
	END_FOR
	
	IF (Parameters.IO.DIn.ResetAlarm OR Parameters.Alarm.Control.ResetAlarms) AND (AlarmA OR AlarmB OR AlarmC) THEN
		IF Parameters.IO.DIn.ResetAlarm THEN
			Main.EventLog.LogEvent(Message := 'Reset alarm via DI', Kind := EventTypes.Information);
		ELSE			
			Main.EventLog.LogEvent(Message := 'Reset alarm via web', Kind := EventTypes.Information);
		END_IF

		FOR N := 0 TO AlarmCount - 1 DO
			TONs[n](IN := FALSE);
		END_FOR
		Latched := NoAlarms;
		Parameters.Alarm.Control.ResetAlarms := FALSE;
		Globals.ResetAlarmsCounter := Globals.ResetAlarmsCounter + 1;
	END_IF
	
	// Transfer from Alarms to Latched according to autoreset and polarity definitions
	LatchedSignalP := ADR(Latched.Signals);
	AutoResetP := ADR(Parameters.Alarm.AutoReset);
	FOR N := 0 TO AlarmCount - 1 DO
		LatchedSignalP^[n] := LatchedSignalP^[n] AND NOT AutoResetP^[n] OR CurrentP^[n];
	END_FOR
	
	// Set parameters alarms
	Parameters.Alarm.Active.A := Latched.Signals.A;
	Parameters.Alarm.Active.B := Latched.Signals.B;
	Parameters.Alarm.Active.C := Latched.Signals.C;
	
	// Set alarms
	AlarmA := NOT AnyEqual(Latched.Signals.A, NoAlarms.Signals.A);
	AlarmB := NOT AnyEqual(Latched.Signals.B, NoAlarms.Signals.B);
	AlarmC := NOT AnyEqual(Latched.Signals.C, NoAlarms.Signals.C);
	AlarmD := FALSE;
	
	CurrentDT := NowDT();
	StartTime();
	IF (CurrentDT <> LastDT) AND (StartTime.ET > LTIME#20S) THEN
		// Add any alarm events to alarm log
		IF (NOT AnyEqual(Latched.Signals, Last.Signals)) or (NOT AnyEqual(Latched.Status, Last.Status)) THEN
			IF NOT Latched.Signals.C.SensorFailure THEN
				LogAlarm(Latched);
			ELSE
				LogAlarmJSON(Item := Latched, VarAdr := ADR(Parameters.IO.Status), VarSize := SIZEOF(Parameters.IO.Status), VarType := 'IoStatus');
			END_IF
			Last := Latched;
		END_IF
		LastDT := CurrentDT;
	END_IF
END_IF

METHOD LogAlarm : BOOL
VAR_INPUT
	Item: AlarmEvent;
END_VAR
VAR
	TempHead, TempTail: INT;
END_VAR
IF __ISVALIDREF(AlarmLogRef) THEN
	TempTail := AlarmLogRef.Tail + 1;
	IF TempTail > Globals.AlarmsHigh THEN
		TempTail := Globals.AlarmsLow;
	END_IF
	
	IF TempTail = AlarmLogRef.Head THEN
		TempHead := AlarmLogRef.Head + 1;
		IF TempHead > Globals.AlarmsHigh THEN
			TempHead := Globals.AlarmsLow;
		END_IF
		AlarmLogRef.Head := TempHead;
	END_IF
	Item.TimeStamp := NowDT();	
	AlarmLogRef.Alarms[AlarmLogRef.Tail] := Item;
	IF IncludeJSON AND (INT_TO_UINT(Len(sJSON)) < SIZEOF(Globals.AlarmLogStrings[AlarmLogRef.Tail]) ) THEN
		Globals.AlarmLogStrings[AlarmLogRef.Tail] := sJSON;
		AlarmLogRef.Alarms[AlarmLogRef.Tail].JSON := TRUE;
	ELSE
		AlarmLogRef.Alarms[AlarmLogRef.Tail].JSON := FALSE;
	END_IF
	
	AlarmLogRef.Tail := TempTail;
	Main.EventLog.LogEventJSON(Message := 'Alarm status changed', Kind := EventTypes.Error, VarAdr := ADR(Item.Signals), VarSize := SIZEOF(Item.Signals), VarType := 'AlarmSignals');
END_IF
END_METHOD

METHOD LogAlarmJSON : BOOL
VAR_INPUT
	Item: AlarmEvent;
	VarType: STRING;
	VarSize: DWORD;
	VarAdr: POINTER TO DWORD;
END_VAR
VAR
	nLen: UDINT;
END_VAR
sJSON := '';
nLen := fbJsonDataType.CopyJsonStringFromSymbol(VarType, VarSize, VarAdr, sJSON,SIZEOF(sJSON));
IncludeJSON := nLen > 0;
LogAlarm(Item := Item);
IncludeJSON := FALSE;
END_METHOD

END_FUNCTION_BLOCK

// ---- DUTs/System/AnyEqual.TcPOU
FUNCTION AnyEqual : BOOL
VAR_INPUT
	A: ANY;
	B: any;
END_VAR
VAR
	bDataTypesEquals: BOOL;
	bDataSizeEquals: BOOL;
	nCount: DINT;
	bDataContentEquals: BOOL;
END_VAR

IF A.TypeClass = B.TypeClass THEN
    bDataTypesEquals := TRUE;
END_IF
IF bDataTypesEquals THEN
    IF (A.diSize = B.diSize) THEN
        bDataSizeEquals := TRUE;
    END_IF
END_IF
IF bDataTypesEquals AND bDataSizeEquals THEN
    // Compare each byte in the ANY-types
	bDataContentEquals := TRUE;
    FOR nCount := 0 TO A.diSize-1 BY 1 DO
        IF A.pValue[nCount] <> B.pValue[nCount] THEN
            bDataContentEquals := FALSE;
            EXIT;
        END_IF
    END_FOR
END_IF
AnyEqual := bDataContentEquals AND bDataSizeEquals AND bDataTypesEquals;

END_FUNCTION

// ---- DUTs/Utilities/Scale.TcPOU
FUNCTION_BLOCK Scale
VAR_INPUT
	EN: BOOL := TRUE;
	x: LREAL;
	x1: LREAL;
	x2: LREAL;
	u1: LREAL;
	u2: LREAL;
END_VAR
VAR_OUTPUT
	ENO: bool;
	u: LREAL;
END_VAR
VAR
END_VAR

IF EN THEN
	IF u1 <= u2 THEN
		u := LimitValue((((x - x1) * (u2 - u1)) / (x2 - x1)) + u1, u1, u2);
	ELSE
		u := LimitValue(u1 - (((x - x1) * (u1 - u2)) / (x2 - x1)), u2, u1);
	END_IF
ELSE
	u := 0;
END_IF
ENO := EN;

END_FUNCTION_BLOCK

// ---- DUTs/Controllers/PidController.TcPOU
FUNCTION_BLOCK PidController
VAR_INPUT
	Param: ControllerParameters;
	EN: BOOL := TRUE;
	SP: LREAL;
	PV: LREAL;
	P: LREAL := 1;
	I: TIME := T#1M;
	Dtime: UDINT;
	DampingTime: TIME;
	SyncCV: LREAL;
	Sync: BOOL;
	Hold: BOOL;
	MinSpeed: LREAL := 0;
	MaxSpeed: LREAL := 1;
END_VAR
VAR_OUTPUT
	CV: LREAL;
	ENO: BOOL;
	Error: LREAL;
END_VAR
VAR
	Ctrl: FB_BA_PIDCtrl;
	TempCV: REAL;
END_VAR

Ctrl(	bEn := EN, 
		rW := LREAL_TO_REAL(SP), 
		rX := LREAL_TO_REAL(PV), 
		rKp := LREAL_TO_REAL(P), 
		udiTn_ms := TIME_TO_UDINT(I), 
		udiTv_ms := Dtime, 
		udiTd_ms := TIME_TO_UDINT(DampingTime), 
		rYMax := TO_REAL(MaxSpeed * 1000), 
		rYMin := TO_REAL(MinSpeed * 1000), 
		rSync := LREAL_TO_REAL(SyncCV * 1000), 
		bSync := Sync, 		
		rY => TempCV, 
		rE => Error
);
CV := TempCV / 1000;
ENO := EN;

END_FUNCTION_BLOCK

// ---- DUTs/Utilities/Average.TcPOU
FUNCTION_BLOCK Average
VAR_INPUT
	NewSample: LREAL;
END_VAR
VAR_OUTPUT
	Value: LREAL;
END_VAR
VAR
	Acc: lreal;
	LastSec: LINT;
END_VAR

IF LastSec = 0 THEN
	Acc := NewSample;
END_IF
IF Globals.SecondsCounter <> LastSec THEN
	Acc := Acc * 0.9;
	Acc := Acc + NewSample;
	Value := Acc / 10;
	LastSec := Globals.SecondsCounter;
END_IF

END_FUNCTION_BLOCK

// ---- DUTs/Utilities/WriteLRealOnlyIf.TcPOU
FUNCTION_BLOCK WriteLRealOnlyIf
VAR_IN_OUT
	Out: LREAL;	
END_VAR
VAR_INPUT
	EN: BOOL := TRUE;
	Value: LREAL;
END_VAR
VAR_OUTPUT
	ENO: bool;
END_VAR
VAR
END_VAR

ENO := EN;
IF EN THEN
	Out := Value;
END_IF

END_FUNCTION_BLOCK

// ---- POUs/SmokeControl.TcPOU
PROGRAM SmokeControl
VAR
	StartupDone: BOOL;
	GreenMasterSmokeControl: GreenMasterSmokeControl; 
	Parameters: REFERENCE TO GreenMasterBaseParameters;
	ParametersFB: REFERENCE TO GreenMasterBaseParametersFB;
	ParametersSC: REFERENCE TO SmokeControlParametersBase;
	ParametersSCFB: REFERENCE TO SmokeControlParametersBaseFB;
	ExerciseTimer: Timer;
	EN: BOOL;
	LocalTime: FB_LocalSystemTime;
	Elapsed: LINT;
	ForceExercise: BOOL;
	Exercising: BOOL;
	CurrentState: INT;
	StateTimer: TImer;
	DetectedDamperError: BOOL;
	DetectedDamperFireAlarm: BOOL;
END_VAR

IF NOT StartupDone THEN
	Parameters REF= Main.GreenMaster.GetParameters();
	ParametersSC REF= Main.GreenMaster.GetParametersSC();
	ParametersFB REF= Main.GreenMaster.GetParametersFB();
	ParametersSCFB REF= Main.GreenMaster.GetParametersSCFB();
	StartupDone := TRUE;
END_IF
EN := GetComponent(Name := ComponentNames.GM_SMOKE_CONTROL).EN;
LocalTime(bEnable := TRUE);
ExerciseTimer(EN := EN);
Elapsed := ExerciseTimer.ElapsedTime();
IF EN AND LocalTime.bValid THEN
	GreenMasterSmokeControl(EN := TRUE, Parameters := Parameters, ParametersSC := ParametersSC);
	GreenMasterSmokeControl.Update(Parameters, ParametersSC, ParametersFB, ParametersSCFB);
END_IF

IF GreenMasterSmokeControl.DamperError AND Parameters.Alarm.Active.B.DamperError THEN
	DetectedDamperError := TRUE;
END_IF
IF DetectedDamperError AND NOT Parameters.Alarm.Active.B.DamperError THEN
	DetectedDamperError := FALSE;
	ForceExercise := TRUE;
END_IF

IF GreenMasterSmokeControl.FireAlarm AND Parameters.Alarm.Active.A.FireLocal THEN
	DetectedDamperFireAlarm := TRUE;
END_IF
IF DetectedDamperFireAlarm AND NOT Parameters.Alarm.Active.A.FireLocal THEN
	DetectedDamperFireAlarm := FALSE;
	GreenMasterSmokeControl.ResetSmokeDetectors := TRUE;
	ForceExercise := TRUE;
END_IF
IF NOT Parameters.Alarm.Status.A.FireLocal THEN
	GreenMasterSmokeControl.ResetSmokeDetectors := FALSE;
END_IF

StateTimer();
CASE CurrentState OF
	0:
		IF EN AND LocalTime.bValid THEN
			IF ((ParametersSC.NetLink.Exercise.Interval > 0) AND (ExerciseTimer.ElapsedTime() > (ParametersSC.NetLink.Exercise.Interval * 3600 * 1000)) AND 
				(
					(WORD_TO_INT(LocalTime.systemTime.wHour) = ParametersSC.NetLink.Exercise.Hour) AND (WORD_TO_INT(LocalTime.systemTime.wMinute) = ParametersSC.NetLink.Exercise.Minute)
				)) OR ForceExercise THEN
				ForceExercise := FALSE;
				Exercising := TRUE;
				StateTimer.Restart();
				CurrentState := 1;
				Main.EventLog.LogEvent(EventTypes.Information, 'Exercising Smoke Control dampers');
			END_IF			
		END_IF
	1:
		IF StateTimer.ElapsedTime() > 10 * 1000 THEN
			GreenMasterSmokeControl.Exercise := TRUE;
			GreenMasterSmokeControl.Write();
			ExerciseTimer.Restart();
			CurrentState := 2;
		END_IF
	2:
		IF StateTimer.ElapsedTime() > 30 * 1000 THEN
			CurrentState := 3;
		END_IF
	3:
		IF (NOT GreenMasterSmokeControl.Exercising) OR (StateTimer.ElapsedTime() > 180 * 1000) THEN
			GreenMasterSmokeControl.Exercise := FALSE;
			Exercising := FALSE;
			CurrentState := 0;
		END_IF
END_CASE

END_PROGRAM

// ---- DUTs/GreenMaster/IO/GreenMasterSmokeControl.TcPOU
FUNCTION_BLOCK GreenMasterSmokeControl extends GreenMasterSmokeControl_Base
VAR_INPUT
	Exercise: BOOL;
	ResetSmokeDetectors: bool;
END_VAR
VAR_OUTPUT
	Exercising: BOOL;
	DamperError: BOOL;
	ServiceAlarm: BOOL;
END_VAR
VAR
	ModbusTCP: ModbusTCP;
	DamperControl: DamperControl;
	DamperModule_0: DamperModule;
	DamperModule_1: DamperModule;
	DamperModule_2: DamperModule;
	DamperModule_3: DamperModule;
	DamperModule_4: DamperModule;
	DamperModule_5: DamperModule;
	DamperModule_6: DamperModule;
	DamperModule_7: DamperModule;
	DamperModule_8: DamperModule;
	DamperModule_9: DamperModule;
	DamperModule_10: DamperModule;
	DamperModule_11: DamperModule;
	DamperModule_12: DamperModule;
	DamperModule_13: DamperModule;
	DamperModule_14: DamperModule;
END_VAR
VAR // added by the converter: edge detectors and wires of the graphical bodies
    _w1, _w2, _w3, _w4 : ANY;
END_VAR


// PAGE Modbus TCP
ModbusTCP(EN := EN, IP := ParametersSC.NetLink.ModbusTCP_IP);
Main.GreenMaster.GetParametersSC().NetLink.Error := ModbusTCP.Error;

// PAGE Smoke Detection
_w1 := DamperModule_0.DamperError OR DamperModule_1.DamperError OR DamperModule_2.DamperError OR DamperModule_3.DamperError OR DamperModule_4.DamperError OR DamperModule_5.DamperError OR DamperModule_6.DamperError OR DamperModule_7.DamperError OR DamperModule_8.DamperError OR DamperModule_9.DamperError OR DamperModule_10.DamperError OR DamperModule_11.DamperError OR DamperModule_12.DamperError OR DamperModule_13.DamperError OR DamperModule_14.DamperError;
DamperModule_4(
    EN := ParametersSC.DamperModules.Unit05.EN,
    UnitID := ParametersSC.DamperModules.Unit05.UnitID,
    ModbusTCP := ModbusTCP,
    Exercise := Exercise,
    ResetSmokeDetector := ResetSmokeDetectors,
    WriteText := ParametersSC.DamperModules.Unit05.Text); // DamperModule
_w2 := DamperModule_0.ServiceAlarm OR DamperModule_1.ServiceAlarm OR DamperModule_2.ServiceAlarm OR DamperModule_3.ServiceAlarm OR DamperModule_4.ServiceAlarm OR DamperModule_5.ServiceAlarm OR DamperModule_6.ServiceAlarm OR DamperModule_7.ServiceAlarm OR DamperModule_8.ServiceAlarm OR DamperModule_9.ServiceAlarm OR DamperModule_10.ServiceAlarm OR DamperModule_11.ServiceAlarm OR DamperModule_12.ServiceAlarm OR DamperModule_13.ServiceAlarm OR DamperModule_14.ServiceAlarm;
DamperModule_5(
    EN := ParametersSC.DamperModules.Unit06.EN,
    UnitID := ParametersSC.DamperModules.Unit06.UnitID,
    ModbusTCP := ModbusTCP,
    Exercise := Exercise,
    ResetSmokeDetector := ResetSmokeDetectors,
    WriteText := ParametersSC.DamperModules.Unit06.Text); // DamperModule
_w3 := DamperModule_0.Exercising OR DamperModule_1.Exercising OR DamperModule_2.Exercising OR DamperModule_3.Exercising OR DamperModule_4.Exercising OR DamperModule_5.Exercising OR DamperModule_6.Exercising OR DamperModule_7.Exercising OR DamperModule_8.Exercising OR DamperModule_9.Exercising OR DamperModule_10.Exercising OR DamperModule_11.Exercising OR DamperModule_12.Fire OR DamperModule_13.Fire OR DamperModule_14.Exercising;
DamperControl(EN := true);
FireAlarm := _w4;
_w4 := DamperModule_0.Fire OR DamperModule_1.Fire OR DamperModule_2.Fire OR DamperModule_3.Fire OR DamperModule_4.Fire OR DamperModule_5.Fire OR DamperModule_6.Fire OR DamperModule_7.Fire OR DamperModule_8.Fire OR DamperModule_9.Fire OR DamperModule_10.Fire OR DamperModule_11.Fire OR DamperModule_12.Fire OR DamperModule_13.Fire OR DamperModule_14.Fire;
Exercising := _w3;
DamperModule_6(
    EN := ParametersSC.DamperModules.Unit07.EN,
    UnitID := ParametersSC.DamperModules.Unit07.UnitID,
    ModbusTCP := ModbusTCP,
    Exercise := Exercise,
    ResetSmokeDetector := ResetSmokeDetectors,
    WriteText := ParametersSC.DamperModules.Unit07.Text); // DamperModule
DamperModule_7(
    EN := ParametersSC.DamperModules.Unit08.EN,
    UnitID := ParametersSC.DamperModules.Unit08.UnitID,
    ModbusTCP := ModbusTCP,
    Exercise := Exercise,
    ResetSmokeDetector := ResetSmokeDetectors,
    WriteText := ParametersSC.DamperModules.Unit08.Text); // DamperModule
DamperModule_8(
    EN := ParametersSC.DamperModules.Unit09.EN,
    UnitID := ParametersSC.DamperModules.Unit09.UnitID,
    ModbusTCP := ModbusTCP,
    Exercise := Exercise,
    ResetSmokeDetector := ResetSmokeDetectors,
    WriteText := ParametersSC.DamperModules.Unit09.Text); // DamperModule
DamperModule_13(
    EN := ParametersSC.DamperModules.Unit14.EN,
    UnitID := ParametersSC.DamperModules.Unit14.UnitID,
    ModbusTCP := ModbusTCP,
    Exercise := Exercise,
    ResetSmokeDetector := ResetSmokeDetectors,
    WriteText := ParametersSC.DamperModules.Unit14.Text); // DamperModule
DamperModule_14(
    EN := ParametersSC.DamperModules.Unit15.EN,
    UnitID := ParametersSC.DamperModules.Unit15.UnitID,
    ModbusTCP := ModbusTCP,
    Exercise := Exercise,
    ResetSmokeDetector := ResetSmokeDetectors,
    WriteText := ParametersSC.DamperModules.Unit15.Text); // DamperModule
DamperModule_11(
    EN := ParametersSC.DamperModules.Unit12.EN,
    UnitID := ParametersSC.DamperModules.Unit12.UnitID,
    ModbusTCP := ModbusTCP,
    Exercise := Exercise,
    ResetSmokeDetector := ResetSmokeDetectors,
    WriteText := ParametersSC.DamperModules.Unit12.Text); // DamperModule
DamperModule_12(
    EN := ParametersSC.DamperModules.Unit13.EN,
    UnitID := ParametersSC.DamperModules.Unit13.UnitID,
    ModbusTCP := ModbusTCP,
    Exercise := Exercise,
    ResetSmokeDetector := ResetSmokeDetectors,
    WriteText := ParametersSC.DamperModules.Unit13.Text); // DamperModule
DamperModule_9(
    EN := ParametersSC.DamperModules.Unit10.EN,
    UnitID := ParametersSC.DamperModules.Unit10.UnitID,
    ModbusTCP := ModbusTCP,
    Exercise := Exercise,
    ResetSmokeDetector := ResetSmokeDetectors,
    WriteText := ParametersSC.DamperModules.Unit10.Text); // DamperModule
DamperModule_10(
    EN := ParametersSC.DamperModules.Unit11.EN,
    UnitID := ParametersSC.DamperModules.Unit11.UnitID,
    ModbusTCP := ModbusTCP,
    Exercise := Exercise,
    ResetSmokeDetector := ResetSmokeDetectors,
    WriteText := ParametersSC.DamperModules.Unit11.Text); // DamperModule
ServiceAlarm := _w2;
DamperModule_2(
    EN := ParametersSC.DamperModules.Unit03.EN,
    UnitID := ParametersSC.DamperModules.Unit03.UnitID,
    ModbusTCP := ModbusTCP,
    Exercise := Exercise,
    ResetSmokeDetector := ResetSmokeDetectors,
    WriteText := ParametersSC.DamperModules.Unit03.Text); // DamperModule
DamperModule_3(
    EN := ParametersSC.DamperModules.Unit04.EN,
    UnitID := ParametersSC.DamperModules.Unit04.UnitID,
    ModbusTCP := ModbusTCP,
    Exercise := Exercise,
    ResetSmokeDetector := ResetSmokeDetectors,
    WriteText := ParametersSC.DamperModules.Unit04.Text); // DamperModule
DamperModule_0(
    EN := ParametersSC.DamperModules.Unit01.EN,
    UnitID := ParametersSC.DamperModules.Unit01.UnitID,
    ModbusTCP := ModbusTCP,
    Exercise := Exercise,
    ResetSmokeDetector := ResetSmokeDetectors,
    WriteText := ParametersSC.DamperModules.Unit01.Text); // DamperModule
DamperModule_1(
    EN := ParametersSC.DamperModules.Unit02.EN,
    UnitID := ParametersSC.DamperModules.Unit02.UnitID,
    ModbusTCP := ModbusTCP,
    Exercise := Exercise,
    ResetSmokeDetector := ResetSmokeDetectors,
    WriteText := ParametersSC.DamperModules.Unit02.Text); // DamperModule
DamperError := _w1;

METHOD Update : BOOL
VAR_INPUT
	Parameters: REFERENCE TO GreenMasterBaseParameters;
	ParametersSC: REFERENCE TO SmokeControlParametersBase;
	ParametersFB: REFERENCE TO GreenMasterBaseParametersFB;
	ParametersSCFB: REFERENCE TO SmokeControlParametersBaseFB;
END_VAR
VAR
	TempAlarm: bool;
END_VAR
ParametersSCFB.NetLink.Update(Parameters);
ParametersSCFB.DamperModules.Unit01.Update(Parameters, DamperModule_0, ParametersSC.DamperModules.Unit01);
ParametersSCFB.DamperModules.Unit02.Update(Parameters, DamperModule_1, ParametersSC.DamperModules.Unit02);
ParametersSCFB.DamperModules.Unit03.Update(Parameters, DamperModule_2, ParametersSC.DamperModules.Unit03);
ParametersSCFB.DamperModules.Unit04.Update(Parameters, DamperModule_3, ParametersSC.DamperModules.Unit04);
ParametersSCFB.DamperModules.Unit05.Update(Parameters, DamperModule_4, ParametersSC.DamperModules.Unit05);
ParametersSCFB.DamperModules.Unit06.Update(Parameters, DamperModule_5, ParametersSC.DamperModules.Unit06);
ParametersSCFB.DamperModules.Unit07.Update(Parameters, DamperModule_6, ParametersSC.DamperModules.Unit07);
ParametersSCFB.DamperModules.Unit08.Update(Parameters, DamperModule_7, ParametersSC.DamperModules.Unit08);
ParametersSCFB.DamperModules.Unit09.Update(Parameters, DamperModule_8, ParametersSC.DamperModules.Unit09);
ParametersSCFB.DamperModules.Unit10.Update(Parameters, DamperModule_9, ParametersSC.DamperModules.Unit10);
ParametersSCFB.DamperModules.Unit11.Update(Parameters, DamperModule_10, ParametersSC.DamperModules.Unit11);
ParametersSCFB.DamperModules.Unit12.Update(Parameters, DamperModule_11, ParametersSC.DamperModules.Unit12);
ParametersSCFB.DamperModules.Unit13.Update(Parameters, DamperModule_12, ParametersSC.DamperModules.Unit13);
ParametersSCFB.DamperModules.Unit14.Update(Parameters, DamperModule_13, ParametersSC.DamperModules.Unit14);
ParametersSCFB.DamperModules.Unit15.Update(Parameters, DamperModule_14, ParametersSC.DamperModules.Unit15);

Parameters.Alarm.Status.B.CommunicationError := (ParametersSC.DamperModules.Unit01.EN AND ParametersSC.DamperModules.Unit01.Error) OR
		(ParametersSC.DamperModules.Unit02.EN AND ParametersSC.DamperModules.Unit02.Error) OR
		(ParametersSC.DamperModules.Unit03.EN AND ParametersSC.DamperModules.Unit03.Error) OR
		(ParametersSC.DamperModules.Unit04.EN AND ParametersSC.DamperModules.Unit04.Error) OR
		(ParametersSC.DamperModules.Unit05.EN AND ParametersSC.DamperModules.Unit05.Error) OR
		(ParametersSC.DamperModules.Unit06.EN AND ParametersSC.DamperModules.Unit06.Error) OR
		(ParametersSC.DamperModules.Unit07.EN AND ParametersSC.DamperModules.Unit07.Error) OR
		(ParametersSC.DamperModules.Unit08.EN AND ParametersSC.DamperModules.Unit08.Error) OR
		(ParametersSC.DamperModules.Unit09.EN AND ParametersSC.DamperModules.Unit09.Error) OR
		(ParametersSC.DamperModules.Unit10.EN AND ParametersSC.DamperModules.Unit10.Error) OR
		(ParametersSC.DamperModules.Unit11.EN AND ParametersSC.DamperModules.Unit11.Error) OR
		(ParametersSC.DamperModules.Unit12.EN AND ParametersSC.DamperModules.Unit12.Error) OR
		(ParametersSC.DamperModules.Unit13.EN AND ParametersSC.DamperModules.Unit13.Error) OR
		(ParametersSC.DamperModules.Unit14.EN AND ParametersSC.DamperModules.Unit14.Error) OR
		(ParametersSC.DamperModules.Unit15.EN AND ParametersSC.DamperModules.Unit15.Error);


Parameters.Alarm.Status.A.FireExtractExternal := ParametersSC.NetLink.Fire.EN AND (
	(ParametersSC.DamperModules.Unit01.EN AND ParametersSC.DamperModules.Unit01.Fire AND ParametersSC.DamperModules.Unit01.CentralFireAlarm) OR
	(ParametersSC.DamperModules.Unit02.EN AND ParametersSC.DamperModules.Unit02.Fire AND ParametersSC.DamperModules.Unit02.CentralFireAlarm) OR
	(ParametersSC.DamperModules.Unit03.EN AND ParametersSC.DamperModules.Unit03.Fire AND ParametersSC.DamperModules.Unit03.CentralFireAlarm) OR
	(ParametersSC.DamperModules.Unit04.EN AND ParametersSC.DamperModules.Unit04.Fire AND ParametersSC.DamperModules.Unit04.CentralFireAlarm) OR
	(ParametersSC.DamperModules.Unit05.EN AND ParametersSC.DamperModules.Unit05.Fire AND ParametersSC.DamperModules.Unit05.CentralFireAlarm) OR
	(ParametersSC.DamperModules.Unit06.EN AND ParametersSC.DamperModules.Unit06.Fire AND ParametersSC.DamperModules.Unit06.CentralFireAlarm) OR
	(ParametersSC.DamperModules.Unit07.EN AND ParametersSC.DamperModules.Unit07.Fire AND ParametersSC.DamperModules.Unit07.CentralFireAlarm) OR
	(ParametersSC.DamperModules.Unit08.EN AND ParametersSC.DamperModules.Unit08.Fire AND ParametersSC.DamperModules.Unit08.CentralFireAlarm) OR
	(ParametersSC.DamperModules.Unit09.EN AND ParametersSC.DamperModules.Unit09.Fire AND ParametersSC.DamperModules.Unit09.CentralFireAlarm) OR
	(ParametersSC.DamperModules.Unit10.EN AND ParametersSC.DamperModules.Unit10.Fire AND ParametersSC.DamperModules.Unit10.CentralFireAlarm) OR
	(ParametersSC.DamperModules.Unit11.EN AND ParametersSC.DamperModules.Unit11.Fire AND ParametersSC.DamperModules.Unit11.CentralFireAlarm) OR
	(ParametersSC.DamperModules.Unit12.EN AND ParametersSC.DamperModules.Unit12.Fire AND ParametersSC.DamperModules.Unit12.CentralFireAlarm) OR
	(ParametersSC.DamperModules.Unit13.EN AND ParametersSC.DamperModules.Unit13.Fire AND ParametersSC.DamperModules.Unit13.CentralFireAlarm) OR
	(ParametersSC.DamperModules.Unit14.EN AND ParametersSC.DamperModules.Unit14.Fire AND ParametersSC.DamperModules.Unit14.CentralFireAlarm) OR
	(ParametersSC.DamperModules.Unit15.EN AND ParametersSC.DamperModules.Unit15.Fire AND ParametersSC.DamperModules.Unit15.CentralFireAlarm));
	
Parameters.Alarm.Status.A.FireLocal := ParametersSC.NetLink.Fire.EN AND (
	(ParametersSC.DamperModules.Unit01.EN AND ParametersSC.DamperModules.Unit01.Fire AND NOT ParametersSC.DamperModules.Unit01.CentralFireAlarm) OR
	(ParametersSC.DamperModules.Unit02.EN AND ParametersSC.DamperModules.Unit02.Fire AND NOT ParametersSC.DamperModules.Unit02.CentralFireAlarm) OR
	(ParametersSC.DamperModules.Unit03.EN AND ParametersSC.DamperModules.Unit03.Fire AND NOT ParametersSC.DamperModules.Unit03.CentralFireAlarm) OR
	(ParametersSC.DamperModules.Unit04.EN AND ParametersSC.DamperModules.Unit04.Fire AND NOT ParametersSC.DamperModules.Unit04.CentralFireAlarm) OR
	(ParametersSC.DamperModules.Unit05.EN AND ParametersSC.DamperModules.Unit05.Fire AND NOT ParametersSC.DamperModules.Unit05.CentralFireAlarm) OR
	(ParametersSC.DamperModules.Unit06.EN AND ParametersSC.DamperModules.Unit06.Fire AND NOT ParametersSC.DamperModules.Unit06.CentralFireAlarm) OR
	(ParametersSC.DamperModules.Unit07.EN AND ParametersSC.DamperModules.Unit07.Fire AND NOT ParametersSC.DamperModules.Unit07.CentralFireAlarm) OR
	(ParametersSC.DamperModules.Unit08.EN AND ParametersSC.DamperModules.Unit08.Fire AND NOT ParametersSC.DamperModules.Unit08.CentralFireAlarm) OR
	(ParametersSC.DamperModules.Unit09.EN AND ParametersSC.DamperModules.Unit09.Fire AND NOT ParametersSC.DamperModules.Unit09.CentralFireAlarm) OR
	(ParametersSC.DamperModules.Unit10.EN AND ParametersSC.DamperModules.Unit10.Fire AND NOT ParametersSC.DamperModules.Unit10.CentralFireAlarm) OR
	(ParametersSC.DamperModules.Unit11.EN AND ParametersSC.DamperModules.Unit11.Fire AND NOT ParametersSC.DamperModules.Unit11.CentralFireAlarm) OR
	(ParametersSC.DamperModules.Unit12.EN AND ParametersSC.DamperModules.Unit12.Fire AND NOT ParametersSC.DamperModules.Unit12.CentralFireAlarm) OR
	(ParametersSC.DamperModules.Unit13.EN AND ParametersSC.DamperModules.Unit13.Fire AND NOT ParametersSC.DamperModules.Unit13.CentralFireAlarm) OR
	(ParametersSC.DamperModules.Unit14.EN AND ParametersSC.DamperModules.Unit14.Fire AND NOT ParametersSC.DamperModules.Unit14.CentralFireAlarm) OR
	(ParametersSC.DamperModules.Unit15.EN AND ParametersSC.DamperModules.Unit15.Fire AND NOT ParametersSC.DamperModules.Unit15.CentralFireAlarm));
END_METHOD

METHOD Write : BOOL
VAR_INPUT
END_VAR
DamperModule_0.StartWrite();
DamperModule_1.StartWrite();
END_METHOD

END_FUNCTION_BLOCK

// ---- DUTs/Smoke Control/DamperControl.TcPOU
FUNCTION_BLOCK DamperControl
VAR_INPUT
	EN: BOOL;
	Interval: TIME;
	StartTime: TIME_OF_DAY;
	AlarmOnlyOnExercise: bool;
END_VAR
VAR_OUTPUT
	ENO: BOOL;
END_VAR
VAR
END_VAR

ENO := EN;

END_FUNCTION_BLOCK

// ---- GVLs/GetComponent.TcPOU
FUNCTION GetComponent : REFERENCE TO Component
VAR_INPUT
	Name: ComponentNames;
END_VAR
VAR
	n: INT;
	Found: int := -1;
	EmptyComponent: Component;
END_VAR

GetComponent REF= EmptyComponent;
FOR n := 0 TO GlobalSettings.MAX_COMPONENTS - 1 DO
	IF GlobalSettings.Components[n].Name = Name THEN
		Found := n;
		EXIT;
	END_IF
END_FOR

IF Found >= 0 THEN
	GetComponent REF= GlobalSettings.Components[Found];
END_IF

END_FUNCTION

// ---- DUTs/Utilities/LREAL_BMUX.TcPOU
FUNCTION LREAL_BMUX : LREAL
VAR_INPUT
	B: BOOL;
	F: LREAL;
	T: LREAL;
END_VAR
VAR
END_VAR

IF NOT B THEN
	LREAL_BMUX := F;
ELSE
	LREAL_BMUX := T;
END_IF

END_FUNCTION

// ---- DUTs/Fans/FanControl.TcPOU
FUNCTION_BLOCK FanControl
VAR_IN_OUT
	Parameters:GreenMasterBaseParameters;
END_VAR
VAR_INPUT
	EN: BOOL;
	ControlMode: FanControlTypes;
	ControlParameters: ControllerParameters;
	Pressure: LREAL;
	PressureError: BOOL;
	Flow: LREAL;
	FlowError: BOOL;
	MasterPV: LREAL;
	FanAlarm: BOOL;
	MinSpeed: LREAL := 0;
	MaxSpeed: LREAL := 1;
	Override: BOOL;
	OverrideCV: LREAL;
	SyncCV: LREAL;
	ExtendedOperation: BOOL;
	PostVentilationTime: TIME := TIME#2M;
	FireExhaust: BOOL;
	FireSupply: BOOL;
	FireExhaustPar: FireParameters;
	FireSupplyPar: FireParameters;
	Damper: BOOL := TRUE;
END_VAR
VAR_OUTPUT
	ENO: BOOL;
	CV: LREAL;
	PV: LREAL;
	FanRunning: BOOL;
	Recirculation: BOOL;
END_VAR
VAR
	Fan: Fan;
	Ramp: Ramp;
	PiController: PidController;
	StartDelay: TON;
	SPC: Interpolate;
	SupplyAirControl: SupplyAirControl;
	MAX_FB_0: MAX_FB;
	MIN_FB_0: MIN_FB;
	TON_0: TON;
	ControlP: LREAL;
	ControlI: TIME;
	ControlSP: LREAL;
	PostVentilation: PostVentilation;
END_VAR
VAR // added by the converter: edge detectors and wires of the graphical bodies
    _w1, _w2, _w4, _w5, _w7 : ANY;
    _w3, _w6 : BOOL;
END_VAR


// PAGE Fan Control
ControlSP := PostVentilation.SP_PostVentilation;
ControlP := ControlParameters.CSP;
ControlI := ControlParameters.P;
PiController(
    Param := ControlParameters,
    EN := _w1,
    SP := ControlSP,
    PV := _w2,
    P := ControlP,
    I := ControlI,
    SyncCV := SyncCV,
    Sync := NOT Override,
    MinSpeed := MinSpeed,
    MaxSpeed := MaxSpeed); // PidController
_w3 := PressureError OR FlowError;
Fan(
    SpeedSP := Ramp.Value,
    EN := _w4,
    Override := Override,
    OverrideCV := OverrideCV,
    MaxSpeed := MaxSpeed,
    MaxSpeedEnabled := TRUE,
    FireExhaust := FireExhaust,
    FireExhaustPar := FireExhaustPar,
    FireSupplyPar := FireSupplyPar,
    FireExhaust := FireExhaust,
    FireSupply := FireSupply);
TON_0(IN := _w3, PT := T#10s); // TON
FanRunning := Fan.Running;
Ramp(EN := _w1, Start := SyncCV, Target := _w5);
CV := Fan.SpeedCV;
_w2 := MUX(ControlMode, Pressure, Flow, MasterPV);
PV := _w2;
_w6 := EN AND NOT FanAlarm AND Damper;
ENO := _w6;
_w4 := _w6 OR Override;
PostVentilation(
    EN := NOT FireExhaust,
    SP := ControlParameters.SP_HighSpeed,
    PostVentilationTime := PostVentilationTime,
    PostVentilationLevel := ControlParameters.SP_HighSpeed);
_w1 := NOT Override AND _w6;
_w7 := LREAL_BMUX(B := (ControlMode = FanControlTypes.Const) and (Parameters.System.Operation.State = SystemStates.Run), F := PiController.CV, T := ControlSP / 100);
_w5 := LREAL_BMUX(B := TON_0.Q, F := _w7, T := 0.5);

END_FUNCTION_BLOCK

// ---- DUTs/Dampers/Damper.TcPOU
FUNCTION_BLOCK Damper EXTENDS BaseDamper
VAR_INPUT
	IO_Open: REFERENCE TO DigitalOutput;
	IO_FB1, IO_FB2: REFERENCE TO DigitalInput;
END_VAR
VAR_OUTPUT
END_VAR
VAR
	DamperMonitor: DamperMonitor; 
	Error: BOOL;
END_VAR

DamperMonitor(Damper := Open, FB1 := IsOpen, FB2 := IsClosed);
Error := DamperMonitor.Error;

END_FUNCTION_BLOCK

// ---- DUTs/Dampers/BaseDamper.TcPOU
FUNCTION_BLOCK BaseDamper
VAR_INPUT
	Open: REFERENCE TO BOOL;
	IsOpen: REFERENCE TO BOOL;
	IsClosed: REFERENCE TO BOOL;
END_VAR
VAR_OUTPUT
END_VAR
VAR
END_VAR

END_FUNCTION_BLOCK

// ---- DUTs/IO/DigitalOutput.TcPOU
FUNCTION_BLOCK DigitalOutput EXTENDS BaseIO
VAR_INPUT
	Value: BOOL;
	Override: BOOL;
	OverrideValue: BOOL;
END_VAR
VAR_OUTPUT
	ProcessValue: BOOL;
	OffTime: LTIME;
	OnTime: LTIME;
END_VAR
VAR
	InitDone: BOOL;
	TempValue: BOOL;
	TimeChange: LTIME;
	LastValue: BOOL;
END_VAR
VAR PERSISTENT
	Inverted: BOOL;
	SavedOverride: BOOL;
	SavedOverrideValue: BOOL;
END_VAR

SUPER^();
IF NOT InitDone THEN
	InitDone := TRUE;
	OverrideValue := SavedOverrideValue;
	Override := SavedOverride;	
	TimeChange := LTIME();
END_IF
SavedOverride := Override;
SavedOverrideValue := OverrideValue;

IF NOT Override THEN
	TempValue := Value;
ELSE
	TempValue := OverrideValue;	
END_IF

IF Inverted THEN
	TempValue := NOT TempValue;
END_IF

ProcessValue := TempValue;

IF ProcessValue <> LastValue THEN
	LastValue := ProcessValue;
	TimeChange := LTIME();
END_IF

IF NOT ProcessValue THEN
	OffTime := LTIME() - TimeChange;
ELSE
	OffTime := LTIME#0S;
END_IF

IF ProcessValue THEN
	OnTime := LTIME() - TimeChange;
ELSE
	OnTime := LTIME#0s;
END_IF

END_FUNCTION_BLOCK

// ---- DUTs/IO/BaseIO.TcPOU
FUNCTION_BLOCK BaseIO
VAR_INPUT
	ProcessError: BOOL;
	ProcessErrorCode: INT := 0;
END_VAR
VAR_OUTPUT
	Error: BOOL;
	ErrorCode: INT := 0;
END_VAR
VAR
	Kind: TIoKind;
END_VAR
VAR PERSISTENT
	{attribute 'TcEncoding':='UTF-8'}
	Category: STRING;
	{attribute 'TcEncoding':='UTF-8'}
	SystemName: STRING;
	{attribute 'TcEncoding':='UTF-8'}
	CustomName: STRING;
	ErrorDescription: STRING;
END_VAR

END_FUNCTION_BLOCK

// ---- DUTs/IO/DigitalInput.TcPOU
FUNCTION_BLOCK DigitalInput EXTENDS BaseIO
VAR_INPUT
	ProcessValue: BOOL;
	Override: BOOL;
	OverrideValue: BOOL;
	Inverted: bool;
END_VAR
VAR_OUTPUT
	Value: BOOL;
END_VAR
VAR
	InitDone: BOOL;
	TempValue: bool;
END_VAR
VAR PERSISTENT
	IsInverted: BOOL;
	SavedOverride: BOOL;
	SavedOverrideValue: BOOL;
END_VAR

SUPER^();
IF NOT InitDone THEN
	InitDone := TRUE;
	OverrideValue := SavedOverrideValue;
	Override := SavedOverride;	
END_IF
IsInverted := Inverted;

SavedOverride := Override;
SavedOverrideValue := OverrideValue;

IF NOT Override THEN
	TempValue := ProcessValue;
ELSE
	TempValue := OverrideValue;	
END_IF

IF IsInverted THEN
	TempValue := NOT TempValue;
END_IF

Value := TempValue;

END_FUNCTION_BLOCK

// ---- DUTs/Dampers/DamperMonitor.TcPOU
FUNCTION_BLOCK DamperMonitor
VAR_INPUT
	Damper: BOOL;	// Damper DO
	FB1: BOOL;		// Open DI
	FB2: BOOL;		// Closed DI
END_VAR
VAR_OUTPUT
	Error: BOOL;
END_VAR
VAR
	DamperSignal: DigitalSignal;
	DamperOpenTimer: Timer;
	DamperClosedTimer: Timer;
END_VAR

DamperSignal(Signal := Damper);
Error := ((DamperSignal.OnTime() > 30000) AND (NOT FB1)) OR
		((DamperSignal.OffTime() > 30000) AND (NOT FB2));

END_FUNCTION_BLOCK

// ---- DUTs/Utilities/DigitalSignal.TcPOU
FUNCTION_BLOCK DigitalSignal
VAR_INPUT
	Signal: BOOL;
END_VAR
VAR_OUTPUT
	State: BOOL;
END_VAR
VAR
	_PosFlank: BOOL;
	_NegFlank: BOOL;
	OffTimer: Timer;
	OnTimer: Timer;
END_VAR

IF Signal <> State THEN
	State := Signal;
	IF State THEN
	  _PosFlank := TRUE;
	ELSE
	  _NegFlank := TRUE;
	END_IF;
END_IF;
IF State THEN
	OffTimer.Restart();
ELSE
	OnTimer.Restart();
END_IF

METHOD NegFlank : BOOL
VAR_INPUT
	Reset: BOOL;
END_VAR
NegFlank := _NegFlank;
if Reset then
	_NegFlank := FALSE;
END_IF
END_METHOD

METHOD OffTime : LINT
VAR_INPUT
END_VAR
IF State THEN
	OffTimer.Restart();
ELSE
	OnTimer.Restart();
END_IF
OffTime := OffTimer.ElapsedTime();
END_METHOD

METHOD OnTime : LINT
VAR_INPUT
END_VAR
IF State THEN
	OffTimer.Restart();
ELSE
	OnTimer.Restart();
END_IF
OnTime := OnTimer.ElapsedTime();
END_METHOD

METHOD PosFlank : BOOL
VAR_INPUT
	Reset: BOOL := FALSE;
END_VAR
PosFlank := _PosFlank;
if Reset then
	_PosFlank := FALSE;
END_IF
END_METHOD

END_FUNCTION_BLOCK

// ---- DUTs/Fans/Fan.TcPOU
FUNCTION_BLOCK Fan
VAR_INPUT
	EN: BOOL;
	SpeedSP: LREAL;
	Override: BOOL;
	OverrideCV: LREAL;
	MaxSpeed: LREAL;
	MaxSpeedEnabled: BOOL := TRUE;
	FireExhaust: BOOL;
	FireSupply: BOOL;
	FireExhaustPar: FireParameters;
	FireSupplyPar: FireParameters;
END_VAR
VAR_OUTPUT
	ENO: BOOL;
	Running: BOOL;
	SpeedCV: LREAL;
	Error: BOOL;
	ErrorCode: INT;
	SpeedError: BOOL;
END_VAR
VAR
	{attribute 'TcEncoding':='UTF-8'}
	ErrorDescription: STRING;
END_VAR
VAR PERSISTENT
	SpeedAlarmDelay: LREAL;
	FanAlarmDelay: LREAL;
	SpeedAlarmAutoReset: BOOL;
	FanAlarmAutoReset: BOOL;
END_VAR

ENO := EN;
Running := EN AND SpeedCV > 0;
IF NOT Override THEN
	IF EN THEN
		SpeedCV := SpeedSP;
	ELSE
		SpeedCV := 0;
	END_IF
ELSE
	SpeedCV := OverrideCV;
END_IF
IF MaxSpeedEnabled AND (SpeedCV > MaxSpeed) and (not Main.GreenMaster.FireAlarm()) THEN
	SpeedCV := MaxSpeed;
END_IF
IF FireExhaust THEN
	IF FireExhaustPar.EN THEN
		SpeedCV := FireExhaustPar.Speed;
	ELSE
		SpeedCV := 0;
	END_IF
ELSif FireSupply then
	IF FireSupplyPar.EN THEN
		SpeedCV := FireSupplyPar.Speed;
	ELSE
		SpeedCV := 0;
	END_IF
END_IF

END_FUNCTION_BLOCK

// ---- DUTs/Controllers/Ramp.TcPOU
FUNCTION_BLOCK Ramp
VAR_INPUT
	EN: BOOL := TRUE;
	Start: LREAL;
	Target: LREAL;
	SpeedUp: LREAL := 0.05;
	SpeedDown: LREAL := 0.2;
END_VAR
VAR_OUTPUT
	ENO: BOOL;
	Value: LREAL;
	Speed: LREAL;
	ElapsedTime: LINT;
END_VAR
VAR
	Timer: Timer;
	LastElapsed: LINT;
	Elapsed: LINT;
	InitDone: BOOL;
END_VAR

IF EN AND InitDone THEN
	Elapsed := Timer.ElapsedTime();
	IF Target >= Start THEN
		Value := MIN(Target, Value + (LINT_TO_LREAL(Elapsed - LastElapsed) / 1000.0) * SpeedUp);
	ELSE
		Value := MAX(Target, Value - (LINT_TO_LREAL(Elapsed - LastElapsed) / 1000.0) * SpeedDown);	
	END_IF
	LastElapsed := Elapsed;
ELSE
	Value := Start;
	Timer.Restart();
	LastElapsed := 0;
	InitDone := TRUE;
END_IF
Elapsed := Timer.ElapsedTime();
ENO := EN;

METHOD Restart : BOOL
VAR_INPUT
	StartValue: LREAL;
END_VAR
Value := StartValue;
Timer.Restart();
LastElapsed := 0;
InitDone := TRUE;
END_METHOD

END_FUNCTION_BLOCK

// ---- DUTs/Controls/SupplyAirControl.TcPOU
FUNCTION_BLOCK SupplyAirControl
VAR_INPUT
	EN: BOOL;
END_VAR
VAR_OUTPUT
	ENO: BOOL;
	Recirculation: BOOL;
END_VAR
VAR
END_VAR

ENO := EN;

END_FUNCTION_BLOCK

// ---- DUTs/Utilities/MAX_FB.TcPOU
FUNCTION_BLOCK MAX_FB
VAR_INPUT
	In1: LREAL;
	In2: LREAL;
END_VAR
VAR_OUTPUT
	Out: LREAL;
END_VAR
VAR
END_VAR

Out := MAX(In1, In2);

END_FUNCTION_BLOCK

// ---- DUTs/Utilities/MIN_FB.TcPOU
FUNCTION_BLOCK MIN_FB
VAR_INPUT
	In1: LREAL;
	In2: LREAL;
END_VAR
VAR_OUTPUT
	Out: LREAL;
END_VAR
VAR
END_VAR

Out := MIN(In1, In2);

END_FUNCTION_BLOCK

// ---- DUTs/Fans/PostVentilation.TcPOU
FUNCTION_BLOCK PostVentilation
VAR_INPUT
	EN: BOOL := TRUE;
	SP: LREAL;
	PostVentilationTime: TIME;
	PostVentilationLevel: LREAL;
END_VAR
VAR_OUTPUT
	ENO: BOOL;
	SP_PostVentilation: LREAL;
END_VAR
VAR
	PostVentilationTOF: TOF;
END_VAR

PostVentilationTOF(IN := SP > 0, PT := PostVentilationTime);
IF EN THEN
	IF PostVentilationTOF.Q THEN
		IF SP > 0 THEN
			SP_PostVentilation := SP;
		ELSE
			SP_PostVentilation := PostVentilationLevel;
		END_IF
	ELSE
		SP_PostVentilation := 0;
	END_IF
ELSE
	SP_PostVentilation := SP;
END_IF

END_FUNCTION_BLOCK

// ---- DUTs/Ventilation/VentilationControl.TcPOU
FUNCTION_BLOCK VentilationControl
VAR_INPUT
	EN: BOOL;
	StopFans: BOOL;
END_VAR
VAR_OUTPUT
	ENO: BOOL;
END_VAR
VAR
END_VAR
VAR PERSISTENT
END_VAR

ENO := EN AND NOT StopFans;

END_FUNCTION_BLOCK

// ---- DUTs/Defrost/Defrost.TcPOU
FUNCTION_BLOCK Defrost
VAR_IN_OUT
	Parameters: GreenMasterBaseParameters;
END_VAR
VAR_INPUT
	EN: BOOL := TRUE;
	Temperature: LREAL := 20;
	Pressure: LREAL;
END_VAR
VAR_OUTPUT
	ENO: BOOL;
	SupplyFlowAdjustment: LREAL;
	ExtractFlowAdjustment: LREAL;
	Damper1: BOOL;
	Damper2: BOOL;
	Damper3: BOOL;
	Damper4: BOOL;
	Damper5: BOOL;
	Damper6: BOOL;
END_VAR
VAR
	DefrostStage: INT;
	DefrostStageTimer: Timer;
	SectionDefrostTimer: Timer;
	SectionToDefrost: DefrostSections;
	Active: BOOL;
	ForceStage2: BOOL;
	ForceStage3: bool;
END_VAR

IF EN THEN
	Active := (Temperature < Parameters.System.Defrost.DefrostTemperature) AND (Parameters.System.Operation.State = SystemStates.Run);
	
	DefrostStageTimer();
	SectionDefrostTimer();
	Parameters.Regulation.SupplyAir.AdjustCSP := SupplyFlowAdjustment;
	Parameters.Regulation.ExtractAir.AdjustCSP := ExtractFlowAdjustment;
	Parameters.System.Defrost.CurrentStage := DefrostStage;
	Parameters.System.Defrost.CurrentSection := SectionToDefrost;
	Parameters.System.Defrost.CurrentTime := TO_LTIME(DefrostStageTimer.ElapsedTime() * 1000000);
	CASE DefrostStage OF
		0:  Parameters.System.Defrost.CurrentPressureLimit := Parameters.System.Defrost.Stage1.PressureLimit;
		1:  Parameters.System.Defrost.CurrentPressureLimit := Parameters.System.Defrost.Stage1.PressureLimit;
		2:  Parameters.System.Defrost.CurrentPressureLimit := Parameters.System.Defrost.Stage2.PressureLimit;
		3:  Parameters.System.Defrost.CurrentPressureLimit := Parameters.System.Defrost.Stage3.PressureLimit;
	END_CASE
	Parameters.System.Defrost.T_QM1_1 := Damper1;
	Parameters.System.Defrost.T_QM1_2 := Damper2;
	Parameters.System.Defrost.T_QM1_3 := Damper3;
	Parameters.System.Defrost.T_QM1_4 := Damper4;
	Parameters.System.Defrost.T_QM1_5 := Damper5;
	Parameters.System.Defrost.T_QM1_6 := Damper6;
	Parameters.System.Defrost.ENO := DefrostStage > 0;
	
	IF Parameters.System.Defrost.EN AND Active THEN
		IF (Pressure >= Parameters.System.Defrost.Stage3.PressureLimit AND 
				Parameters.System.Defrost.Stage3.EN AND
				DefrostStage < 3) OR ForceStage3 THEN
			ForceStage3 := FALSE;		
			SupplyFlowAdjustment := Parameters.System.Defrost.Stage3.SupplyAir;
			ExtractFlowAdjustment := Parameters.System.Defrost.Stage3.ExtractAir;
			DefrostStage := 3;
			SectionToDefrost := 11;
			DefrostStageTimer.Restart();
		ELSIF (Pressure >= Parameters.System.Defrost.Stage2.PressureLimit AND 
				Parameters.System.Defrost.Stage2.EN AND
				DefrostStage < 2) OR ForceStage2 THEN	
			ForceStage2 := FALSE;	
			SupplyFlowAdjustment := Parameters.System.Defrost.Stage2.SupplyAir;
			ExtractFlowAdjustment := Parameters.System.Defrost.Stage2.ExtractAir;
			DefrostStage := 2;
			SectionToDefrost := 7;
			DefrostStageTimer.Restart();
		ELSIF Pressure >= Parameters.System.Defrost.Stage1.PressureLimit AND 
				Parameters.System.Defrost.Stage1.EN AND
				DefrostStage < 1 THEN		
			SupplyFlowAdjustment := Parameters.System.Defrost.Stage1.SupplyAir;
			ExtractFlowAdjustment := Parameters.System.Defrost.Stage1.ExtractAir;
			DefrostStage := 1;
			SectionToDefrost := 1;
			DefrostStageTimer.Restart();
		END_IF
		
		IF DefrostStage = 0 THEN
			SupplyFlowAdjustment := 1;
			ExtractFlowAdjustment := 1;		
		END_IF
		
		Damper1 := Parameters.System.Defrost.Sections >= 1;
		Damper2 := Parameters.System.Defrost.Sections >= 2;
		Damper3 := Parameters.System.Defrost.Sections >= 3;
		Damper4 := Parameters.System.Defrost.Sections >= 4;
		Damper5 := Parameters.System.Defrost.Sections >= 5;
		Damper6 := Parameters.System.Defrost.Sections >= 6;
		IF DefrostStage > 0 THEN
			CASE SectionToDefrost OF
				// Close one at a time
				DefrostSections.S1: Damper1 := FALSE;
				DefrostSections.S2: Damper2 := FALSE;
				DefrostSections.S3: Damper3 := FALSE;
				DefrostSections.S4: Damper4 := FALSE;
				DefrostSections.S5: Damper5 := FALSE;
				DefrostSections.S6: Damper6 := FALSE;
				DefrostSections.S1_3: Damper1 := FALSE; Damper3 := FALSE;
				DefrostSections.S2_4: Damper2 := FALSE; Damper4 := FALSE;
				DefrostSections.S3_5: Damper3 := FALSE; Damper5 := FALSE;
				DefrostSections.S4_6: Damper4 := FALSE; Damper6 := FALSE;
				DefrostSections.S1_3_5: Damper1 := FALSE; Damper3 := FALSE; Damper5 := FALSE;
				DefrostSections.S2_4_6: Damper2 := FALSE; Damper4 := FALSE; Damper6 := FALSE;
			END_CASE
			
			IF (SectionToDefrost > 0) AND (SectionDefrostTimer.ET > TO_LTIME(Parameters.System.Defrost.SectionTime)) THEN
				SectionDefrostTimer.Restart();
				// Next section
				IF DefrostStage = 1 THEN	
					CASE SectionToDefrost OF
						1:
							IF Parameters.System.Defrost.Sections > 1 THEN
								SectionToDefrost := 2;
							ELSE
								SectionToDefrost := 0;
							END_IF
						2:
							IF Parameters.System.Defrost.Sections > 2 THEN
								SectionToDefrost := 3;
							ELSE
								SectionToDefrost := 0;
							END_IF
						3:
							IF Parameters.System.Defrost.Sections > 3 THEN
								SectionToDefrost := 4;
							ELSE
								SectionToDefrost := 0;
							END_IF
						4:
							IF Parameters.System.Defrost.Sections > 4 THEN
								SectionToDefrost := 5;
							ELSE
								SectionToDefrost := 0;
							END_IF
						5:
							IF Parameters.System.Defrost.Sections > 5 THEN
								SectionToDefrost := 6;
							ELSE
								SectionToDefrost := 0;
							END_IF
						ELSE
							SectionToDefrost := DefrostSections.S0;
					END_CASE
					IF( SectionToDefrost = 0) AND (Pressure >= Parameters.System.Defrost.Stage1.PressureLimit) THEN
						ForceStage2 := TRUE;
					END_IF
				ELSIF DefrostStage = 2 THEN	
					CASE SectionToDefrost OF
						7:
							IF Parameters.System.Defrost.Sections > 2 THEN
								SectionToDefrost := 8;
							ELSE
								SectionToDefrost := 0;
							END_IF
						8: 
							IF Parameters.System.Defrost.Sections > 4 THEN
								SectionToDefrost := 9;
							ELSE
								SectionToDefrost := 0;
							END_IF
						9: 
							IF Parameters.System.Defrost.Sections > 4 THEN
								SectionToDefrost := 10;
							ELSE
								SectionToDefrost := 0;
							END_IF
						ELSE
							SectionToDefrost := 0;
					END_CASE
					IF( SectionToDefrost = 0) AND (Pressure >= Parameters.System.Defrost.Stage2.PressureLimit) THEN
						ForceStage3 := TRUE;
					END_IF
				ELSIF DefrostStage = 3 THEN
					CASE SectionToDefrost OF
						11:
							SectionToDefrost := 12;
						ELSE
							SectionToDefrost := 0;
					end_case
				END_IF
				SectionDefrostTimer.Restart(); // Reinit Section defrost interval
			END_IF
		ELSE
			SectionToDefrost := 0;
		END_IF
		IF SectionToDefrost = 0 THEN
			DefrostStage := 0;
		END_IF
	ELSE
		SupplyFlowAdjustment := 1.0;
		ExtractFlowAdjustment := 1.0;
		DefrostStage := 0;
		SectionToDefrost := 0;
		SectionDefrostTimer.Restart();
		DefrostStageTimer.Restart();
		
		Damper1 := (Parameters.System.Defrost.Sections >= 1) AND (Parameters.System.Operation.State <> SystemStates.Idle);
		Damper2 := (Parameters.System.Defrost.Sections >= 2) AND (Parameters.System.Operation.State <> SystemStates.Idle);
		Damper3 := (Parameters.System.Defrost.Sections >= 3) AND (Parameters.System.Operation.State <> SystemStates.Idle);
		Damper4 := (Parameters.System.Defrost.Sections >= 4) AND (Parameters.System.Operation.State <> SystemStates.Idle);
		Damper5 := (Parameters.System.Defrost.Sections >= 5) AND (Parameters.System.Operation.State <> SystemStates.Idle);
		Damper6 := (Parameters.System.Defrost.Sections >= 6) AND (Parameters.System.Operation.State <> SystemStates.Idle);
		
	END_IF
	Parameters.IO.DOut.T_QM1_1 := Damper1;
	Parameters.IO.DOut.T_QM1_2 := Damper2;
	Parameters.IO.DOut.T_QM1_3 := Damper3;
	Parameters.IO.DOut.T_QM1_4 := Damper4;
	Parameters.IO.DOut.T_QM1_5 := Damper5;
	Parameters.IO.DOut.T_QM1_6 := Damper6;
END_IF

END_FUNCTION_BLOCK

// ---- DUTs/Utilities/WriteLRealIf.TcPOU
FUNCTION_BLOCK WriteLRealIf
VAR_IN_OUT
	Out: LREAL;
END_VAR
VAR_INPUT
	EN: BOOL := TRUE;
	In: LREAL;
END_VAR
VAR_OUTPUT
	ENO: bool;
END_VAR
VAR
END_VAR

ENO := EN;
IF EN THEN
	Out := In;
ELSE
	Out := 0.0;	
END_IF

END_FUNCTION_BLOCK

// ---- DUTs/Custom/_Standard/Standard_Interface.TcPOU
FUNCTION_BLOCK Standard_Interface
VAR_INPUT
	AIn: REFERENCE TO AnalogInputs;
	EN: BOOL;
END_VAR
VAR_OUTPUT
	ENO: BOOL;
END_VAR
VAR
	InitDone: BOOL;
	PreEN: bool;
	Parameters: REFERENCE TO GreenMasterBaseParameters;
	ParametersSC: REFERENCE TO SmokeControlParametersBase;
	GM_XXL: REFERENCE TO GreenMasterXXL_FB;
	T_BT1, T_BT2, T_BT3, H_BT1, F_BT2: TemperatureInput;
	bTemp: BOOL;
	rTemp: REAL;
	lrTemp: LREAL;
	tTemp: TIME;
	ltTemp: LTIME;
	modeTemp: FanControlTypes;
	FirstTime: BOOL;
	TimeChannelActive: BOOL;
	TimeChannelEnabled: BOOL;
	n: UINT;
	TimeChannelFallback: TimeChannel1CH;
	TimeChannelFallback_Data: TimeChannel1CH_Data;
	WatchdogTOF: TOF;
	LastWatchDog: INT;
	SetPointAdjustment: SetPointAdjustment;
	CurrentPV: LREAL;
	
	SavedDisabledStates: AlarmSignals;
	AlarmSignalsTrueExceptFirePanel: AlarmSignals;
	StatusP: POINTER TO ARRAY [0..SIZEOF(AlarmSignals) - 1] OF BOOL;
	AlarmCount: UINT := SIZEOF(AlarmSignals);
	ResetAlarmTON: TON;
	SavedParameters: GreenMasterBaseParameters;
	SavedInterface: GreenMasterSettings;
	SavedParametersSC: SmokeControlParametersBase;
	TestExchange: BOOL := FALSE;
	UpdateTON: TON;
END_VAR

IF NOT InitDone THEN
	Parameters REF= Main.GreenMaster.GetParameters();
	ParametersSC REF= Main.GreenMaster.GetParametersSC();
	GM_XXL REF= Main.GreenMaster;
	SavedParameters := Parameters;
	SavedInterface := ADS_Standard.Tags.Settings;
	SavedParametersSC := ParametersSC;
	InitDone := TRUE;
END_IF;

TimeChannelEnabled := FALSE;
TimeChannelActive := FALSE;
WatchdogTOF(IN := (NOT ADS_Standard.Tags.Settings.WatchdogEnabled) OR (ADS_Standard.Tags.Settings.Watchdog <> LastWatchDog), PT := T#5M);

IF WatchdogTOF.Q THEN
	ENO := EN AND (ADS_Standard.Tags.Settings.RemoteStart > 0) AND TimeChannelEnabled AND TimeChannelActive;
ELSE
	ENO := EN AND (ADS_Standard.Tags.Settings.RemoteStart > 0) AND TimeChannelFallback_Data.Q;
END_IF

IF EN THEN
	
	Globals.IO.DOut.DO16 := ADS_Standard.Tags.Status.C_GP1_CMD;
	UpdateTON(IN := TRUE, PT := T#1S);
	// --------------------------------------------------------------------------------
	// Transfer from Standard tags to settings
	IF Parameters.System.Operation.RemoteEN AND UpdateTON.Q THEN
		UpdateTON(IN := False);
		ExchangeData(	ADR(Parameters.Regulation.NightCoolingRequest), 
						ADR(ADS_Standard.Tags.Settings.NightCoolingEN), 
						SIZEOF(Parameters.Regulation.NightCoolingRequest), 
						ADR(SavedParameters.Regulation.NightCoolingRequest), 
						ADR(SavedInterface.NightCoolingEN), 
						'BOOL', ('Parameters.Regulation.NightCoolingRequest'), ('NightCoolingEN'));	
		ExchangeData(	ADR(Parameters.Alarm.Control.ResetAlarms), 
						ADR(ADS_Standard.Tags.Settings.ResetAlarms), 
						SIZEOF(Parameters.Alarm.Control.ResetAlarms), 
						ADR(SavedParameters.Alarm.Control.ResetAlarms), 
						ADR(SavedInterface.ResetAlarms), 
						'BOOL', 'Parameters.Alarm.Control.ResetAlarms', 'ResetAlarms');	
		ResetAlarmTON(IN := ADS_Standard.Tags.Settings.ResetAlarms, PT := T#3S);
		IF ResetAlarmTON.Q THEN
			ADS_Standard.Tags.Settings.ResetAlarms := FALSE;
		END_IF
		ExchangeData(	ADR(Parameters.Regulation.Control.EN), 
						ADR(ADS_Standard.Tags.Settings.VentilationEN), 
						SIZEOF(Parameters.Regulation.Control.EN), 
						ADR(SavedParameters.Regulation.Control.EN), 
						ADR(SavedInterface.VentilationEN), 
						'BOOL', ('Parameters.Regulation.Control.EN'), ('VentilationEN'));	
		ExchangeData(	ADR(Parameters.Regulation.Temperature.EN), 
						ADR(ADS_Standard.Tags.Settings.TemperatureControlEN), 
						SIZEOF(Parameters.Regulation.Temperature.EN), 
						ADR(SavedParameters.Regulation.Temperature.EN), 
						ADR(SavedInterface.TemperatureControlEN), 
						'BOOL', ('Parameters.Regulation.Temperature.EN'), ('ADS TemperatureControlEN'));	
		ExchangeData(	ADR(Parameters.Regulation.Temperature.TemperatureControlSource), 
						ADR(ADS_Standard.Tags.Settings.TemperatureControlPV), 
						SIZEOF(Parameters.Regulation.Temperature.TemperatureControlSource), 
						ADR(SavedParameters.Regulation.Temperature.TemperatureControlSource), 
						ADR(SavedInterface.TemperatureControlPV), 
						'INT', ('Parameters.Regulation.Temperature.TemperatureControlSource'), ('ADS TemperatureControlPV'));	
		
		ExchangeData(	ADR(Parameters.Regulation.Temperature.Control.SP), 
						ADR(ADS_Standard.Tags.Settings.Temperature_SP), 
						SIZEOF(Parameters.Regulation.Temperature.Control.SP), 
						ADR(SavedParameters.Regulation.Temperature.Control.SP), 
						ADR(SavedInterface.Temperature_SP), 
						'LREAL', ('Parameters.Regulation.Temperature.Control.SP'), ('Temperature_SP'));	
		ExchangeData(	ADR(Parameters.Regulation.Temperature.SetPointAdjustment.Curve), 
						ADR(ADS_Standard.Tags.Settings.T_BT1_CURVE), 
						SIZEOF(Parameters.Regulation.Temperature.SetPointAdjustment.Curve), 
						ADR(SavedParameters.Regulation.Temperature.SetPointAdjustment.Curve), 
						ADR(SavedInterface.T_BT1_CURVE), 
						'SetPointOffsetCurve', ('Parameters.Regulation.Temperature.SetPointAdjustment.Curve'), ('SetPointOffsetCurve'));	
		ExchangeData(	ADR(Parameters.Alarm.Delay.B.HeatExchangerEfficiency), 
						ADR(ADS_Standard.Tags.Settings.TX1_EFF_AD), 
						SIZEOF(Parameters.Alarm.Delay.B.HeatExchangerEfficiency), 
						ADR(SavedParameters.Alarm.Delay.B.HeatExchangerEfficiency), 
						ADR(SavedInterface.TX1_EFF_AD), 
						'TIME', ('Parameters.Alarm.Delay.B.HeatExchangerEfficiency'), ('HeatExchangerEfficiencyAlarmDelay'));	
		ExchangeData(	ADR(Parameters.Alarm.Limits.B.HeatExchangerEfficiency), 
						ADR(ADS_Standard.Tags.Settings.TX1_EFF_ALL), 
						SIZEOF(Parameters.Alarm.Limits.B.HeatExchangerEfficiency), 
						ADR(SavedParameters.Alarm.Limits.B.HeatExchangerEfficiency), 
						ADR(SavedInterface.TX1_EFF_ALL), 
						'REAL', ('Parameters.Alarm.Limits.B.HeatExchangerEfficiency'), ('HeatExchangerEfficiencyAlarmLimit'));	
		
		ExchangeData_LREAL_REAL(	ADR(Parameters.Regulation.Temperature.Control.P), 
						ADR(ADS_Standard.Tags.Settings.TemperatureControl_P), 
						ADR(SavedParameters.Regulation.Temperature.Control.P), 
						ADR(SavedInterface.TemperatureControl_P), 
						('Parameters.Regulation.Temperature.Control.P'), ('TemperatureControl_P'));	

		ExchangeData(	ADR(Parameters.Regulation.Temperature.Control.I), 
						ADR(ADS_Standard.Tags.Settings.TemperatureControl_I), 
						SIZEOF(Parameters.Regulation.Temperature.Control.I),
						ADR(SavedParameters.Regulation.Temperature.Control.I), 
						ADR(SavedInterface.TemperatureControl_I), 
						'TIME', ('Parameters.Regulation.Temperature.Control.I'), ('TemperatureControl_I'));	


		ExchangeData(	ADR(Parameters.Regulation.Temperature.Control.D), 
						ADR(ADS_Standard.Tags.Settings.TemperatureControl_D), 
						SIZEOF(Parameters.Regulation.Temperature.Control.D),
						ADR(SavedParameters.Regulation.Temperature.Control.D), 
						ADR(SavedInterface.TemperatureControl_D), 
						'TIME', ('Parameters.Regulation.Temperature.Control.D'), ('TemperatureControl_D'));	

		ExchangeData(	ADR(Parameters.System.Operation.StartupHeatRecoveryTime), 
						ADR(ADS_Standard.Tags.Settings.StartupHeatRecoveryTime), 
						SIZEOF(Parameters.System.Operation.StartupHeatRecoveryTime),
						ADR(SavedParameters.System.Operation.StartupHeatRecoveryTime), 
						ADR(SavedInterface.StartupHeatRecoveryTime), 
						'TIME', ('Parameters.System.Operation.StartupHeatRecoveryTime'), ('StartupHeatRecoveryTime'));	


		//Parameters.System.Operation.StartupHeatRecoveryTime := TIME_TO_LTIME(ADS_Standard.Tags.Settings.StartupHeatRecoveryTime);
		//Parameters.System.Operation.PostFireVentilationTime := TIME_TO_LTIME(ADS_Standard.Tags.Settings.PostFireVentilationTime);
		
		ExchangeData(	ADR(Parameters.System.Operation.TimeChannels.TC01.OffTime), 
						ADR(ADS_Standard.Tags.Settings.TC.CF1), 
						SIZEOF(Parameters.System.Operation.TimeChannels.TC01.OffTime), 
						ADR(SavedParameters.System.Operation.TimeChannels.TC01.OffTime), 
						ADR(SavedInterface.TC.CF1), 
						'UINT', ('Parameters.System.Operation.TimeChannels.TC01.OffTime'), ('CF1'));	
		ExchangeData(	ADR(Parameters.System.Operation.TimeChannels.TC02.OffTime), 
						ADR(ADS_Standard.Tags.Settings.TC.CF2), 
						SIZEOF(Parameters.System.Operation.TimeChannels.TC02.OffTime), 
						ADR(SavedParameters.System.Operation.TimeChannels.TC02.OffTime), 
						ADR(SavedInterface.TC.CF2), 
						'UINT', ('Parameters.System.Operation.TimeChannels.TC02.OffTime'), ('CF2'));	
		ExchangeData(	ADR(Parameters.System.Operation.TimeChannels.TC03.OffTime), 
						ADR(ADS_Standard.Tags.Settings.TC.CF3), 
						SIZEOF(Parameters.System.Operation.TimeChannels.TC03.OffTime), 
						ADR(SavedParameters.System.Operation.TimeChannels.TC03.OffTime), 
						ADR(SavedInterface.TC.CF3), 
						'UINT', ('Parameters.System.Operation.TimeChannels.TC03.OffTime'), ('CF3'));	
		ExchangeData(	ADR(Parameters.System.Operation.TimeChannels.TC04.OffTime), 
						ADR(ADS_Standard.Tags.Settings.TC.CF4), 
						SIZEOF(Parameters.System.Operation.TimeChannels.TC04.OffTime), 
						ADR(SavedParameters.System.Operation.TimeChannels.TC04.OffTime), 
						ADR(SavedInterface.TC.CF4), 
						'UINT', ('Parameters.System.Operation.TimeChannels.TC04.OffTime'), ('CF4'));	
		ExchangeData(	ADR(Parameters.System.Operation.TimeChannels.TC05.OffTime), 
						ADR(ADS_Standard.Tags.Settings.TC.CF5), 
						SIZEOF(Parameters.System.Operation.TimeChannels.TC05.OffTime), 
						ADR(SavedParameters.System.Operation.TimeChannels.TC05.OffTime), 
						ADR(SavedInterface.TC.CF5), 
						'UINT', ('Parameters.System.Operation.TimeChannels.TC05.OffTime'), ('CF5'));	
		ExchangeData(	ADR(Parameters.System.Operation.TimeChannels.TC06.OffTime), 
						ADR(ADS_Standard.Tags.Settings.TC.CF6), 
						SIZEOF(Parameters.System.Operation.TimeChannels.TC06.OffTime), 
						ADR(SavedParameters.System.Operation.TimeChannels.TC06.OffTime), 
						ADR(SavedInterface.TC.CF6), 
						'UINT', ('Parameters.System.Operation.TimeChannels.TC06.OffTime'), ('CF6'));	
		ExchangeData(	ADR(Parameters.System.Operation.TimeChannels.TC07.OffTime), 
						ADR(ADS_Standard.Tags.Settings.TC.CF7), 
						SIZEOF(Parameters.System.Operation.TimeChannels.TC07.OffTime), 
						ADR(SavedParameters.System.Operation.TimeChannels.TC07.OffTime), 
						ADR(SavedInterface.TC.CF7), 
						'UINT', ('Parameters.System.Operation.TimeChannels.TC07.OffTime'), ('CF7'));	

		ExchangeData(	ADR(Parameters.System.Operation.TimeChannels.TC11.OffTime), 
						ADR(ADS_Standard.Tags.Settings.TC.CF11), 
						SIZEOF(Parameters.System.Operation.TimeChannels.TC11.OffTime), 
						ADR(SavedParameters.System.Operation.TimeChannels.TC11.OffTime), 
						ADR(SavedInterface.TC.CF11), 
						'UINT', ('Parameters.System.Operation.TimeChannels.TC11.OffTime'), ('CF11'));	
		ExchangeData(	ADR(Parameters.System.Operation.TimeChannels.TC12.OffTime), 
						ADR(ADS_Standard.Tags.Settings.TC.CF12), 
						SIZEOF(Parameters.System.Operation.TimeChannels.TC12.OffTime), 
						ADR(SavedParameters.System.Operation.TimeChannels.TC12.OffTime), 
						ADR(SavedInterface.TC.CF12), 
						'UINT', ('Parameters.System.Operation.TimeChannels.TC12.OffTime'), ('CF12'));	
		ExchangeData(	ADR(Parameters.System.Operation.TimeChannels.TC13.OffTime), 
						ADR(ADS_Standard.Tags.Settings.TC.CF13), 
						SIZEOF(Parameters.System.Operation.TimeChannels.TC13.OffTime), 
						ADR(SavedParameters.System.Operation.TimeChannels.TC13.OffTime), 
						ADR(SavedInterface.TC.CF13), 
						'UINT', ('Parameters.System.Operation.TimeChannels.TC13.OffTime'), ('CF13'));	
		ExchangeData(	ADR(Parameters.System.Operation.TimeChannels.TC14.OffTime), 
						ADR(ADS_Standard.Tags.Settings.TC.CF14), 
						SIZEOF(Parameters.System.Operation.TimeChannels.TC14.OffTime), 
						ADR(SavedParameters.System.Operation.TimeChannels.TC14.OffTime), 
						ADR(SavedInterface.TC.CF14), 
						'UINT', ('Parameters.System.Operation.TimeChannels.TC14.OffTime'), ('CF14'));	
		ExchangeData(	ADR(Parameters.System.Operation.TimeChannels.TC15.OffTime), 
						ADR(ADS_Standard.Tags.Settings.TC.CF15), 
						SIZEOF(Parameters.System.Operation.TimeChannels.TC15.OffTime), 
						ADR(SavedParameters.System.Operation.TimeChannels.TC15.OffTime), 
						ADR(SavedInterface.TC.CF15), 
						'UINT', ('Parameters.System.Operation.TimeChannels.TC15.OffTime'), ('CF15'));	
		ExchangeData(	ADR(Parameters.System.Operation.TimeChannels.TC16.OffTime), 
						ADR(ADS_Standard.Tags.Settings.TC.CF16), 
						SIZEOF(Parameters.System.Operation.TimeChannels.TC16.OffTime), 
						ADR(SavedParameters.System.Operation.TimeChannels.TC16.OffTime), 
						ADR(SavedInterface.TC.CF16), 
						'UINT', ('Parameters.System.Operation.TimeChannels.TC16.OffTime'), ('CF16'));	
		ExchangeData(	ADR(Parameters.System.Operation.TimeChannels.TC17.OffTime), 
						ADR(ADS_Standard.Tags.Settings.TC.CF17), 
						SIZEOF(Parameters.System.Operation.TimeChannels.TC17.OffTime), 
						ADR(SavedParameters.System.Operation.TimeChannels.TC17.OffTime), 
						ADR(SavedInterface.TC.CF17), 
						'UINT', ('Parameters.System.Operation.TimeChannels.TC17.OffTime'), ('CF17'));	

		ExchangeData(	ADR(Parameters.System.Operation.TimeChannels.TC21.OffTime), 
						ADR(ADS_Standard.Tags.Settings.TC.CF21), 
						SIZEOF(Parameters.System.Operation.TimeChannels.TC21.OffTime), 
						ADR(SavedParameters.System.Operation.TimeChannels.TC21.OffTime), 
						ADR(SavedInterface.TC.CF21), 
						'UINT', ('Parameters.System.Operation.TimeChannels.TC21.OffTime'), ('CF21'));	
		ExchangeData(	ADR(Parameters.System.Operation.TimeChannels.TC22.OffTime), 
						ADR(ADS_Standard.Tags.Settings.TC.CF22), 
						SIZEOF(Parameters.System.Operation.TimeChannels.TC22.OffTime), 
						ADR(SavedParameters.System.Operation.TimeChannels.TC22.OffTime), 
						ADR(SavedInterface.TC.CF22), 
						'UINT', ('Parameters.System.Operation.TimeChannels.TC22.OffTime'), ('CF22'));	
		ExchangeData(	ADR(Parameters.System.Operation.TimeChannels.TC23.OffTime), 
						ADR(ADS_Standard.Tags.Settings.TC.CF23), 
						SIZEOF(Parameters.System.Operation.TimeChannels.TC23.OffTime), 
						ADR(SavedParameters.System.Operation.TimeChannels.TC23.OffTime), 
						ADR(SavedInterface.TC.CF23), 
						'UINT', ('Parameters.System.Operation.TimeChannels.TC23.OffTime'), ('CF23'));	
		ExchangeData(	ADR(Parameters.System.Operation.TimeChannels.TC24.OffTime), 
						ADR(ADS_Standard.Tags.Settings.TC.CF24), 
						SIZEOF(Parameters.System.Operation.TimeChannels.TC24.OffTime), 
						ADR(SavedParameters.System.Operation.TimeChannels.TC24.OffTime), 
						ADR(SavedInterface.TC.CF24), 
						'UINT', ('Parameters.System.Operation.TimeChannels.TC24.OffTime'), ('CF24'));	
		ExchangeData(	ADR(Parameters.System.Operation.TimeChannels.TC25.OffTime), 
						ADR(ADS_Standard.Tags.Settings.TC.CF25), 
						SIZEOF(Parameters.System.Operation.TimeChannels.TC25.OffTime), 
						ADR(SavedParameters.System.Operation.TimeChannels.TC25.OffTime), 
						ADR(SavedInterface.TC.CF25), 
						'UINT', ('Parameters.System.Operation.TimeChannels.TC25.OffTime'), ('CF25'));	
		ExchangeData(	ADR(Parameters.System.Operation.TimeChannels.TC26.OffTime), 
						ADR(ADS_Standard.Tags.Settings.TC.CF26), 
						SIZEOF(Parameters.System.Operation.TimeChannels.TC26.OffTime), 
						ADR(SavedParameters.System.Operation.TimeChannels.TC26.OffTime), 
						ADR(SavedInterface.TC.CF26), 
						'UINT', ('Parameters.System.Operation.TimeChannels.TC26.OffTime'), ('CF26'));	
		ExchangeData(	ADR(Parameters.System.Operation.TimeChannels.TC27.OffTime), 
						ADR(ADS_Standard.Tags.Settings.TC.CF27), 
						SIZEOF(Parameters.System.Operation.TimeChannels.TC27.OffTime), 
						ADR(SavedParameters.System.Operation.TimeChannels.TC27.OffTime), 
						ADR(SavedInterface.TC.CF27), 
						'UINT', ('Parameters.System.Operation.TimeChannels.TC27.OffTime'), ('CF27'));	

		ExchangeData(	ADR(Parameters.System.Operation.TimeChannels.TC01.OnTime), 
						ADR(ADS_Standard.Tags.Settings.TC.CT1), 
						SIZEOF(Parameters.System.Operation.TimeChannels.TC01.OnTime), 
						ADR(SavedParameters.System.Operation.TimeChannels.TC01.OnTime), 
						ADR(SavedInterface.TC.CT1), 
						'UINT', ('Parameters.System.Operation.TimeChannels.TC01.OnTime'), ('CT1'));	
		ExchangeData(	ADR(Parameters.System.Operation.TimeChannels.TC02.OnTime), 
						ADR(ADS_Standard.Tags.Settings.TC.CT2), 
						SIZEOF(Parameters.System.Operation.TimeChannels.TC02.OnTime), 
						ADR(SavedParameters.System.Operation.TimeChannels.TC02.OnTime), 
						ADR(SavedInterface.TC.CT2), 
						'UINT', ('Parameters.System.Operation.TimeChannels.TC02.OnTime'), ('CT2'));	
		ExchangeData(	ADR(Parameters.System.Operation.TimeChannels.TC03.OnTime), 
						ADR(ADS_Standard.Tags.Settings.TC.CT3), 
						SIZEOF(Parameters.System.Operation.TimeChannels.TC03.OnTime), 
						ADR(SavedParameters.System.Operation.TimeChannels.TC03.OnTime), 
						ADR(SavedInterface.TC.CT3), 
						'UINT', ('Parameters.System.Operation.TimeChannels.TC03.OnTime'), ('CT3'));	
		ExchangeData(	ADR(Parameters.System.Operation.TimeChannels.TC04.OnTime), 
						ADR(ADS_Standard.Tags.Settings.TC.CT4), 
						SIZEOF(Parameters.System.Operation.TimeChannels.TC04.OnTime), 
						ADR(SavedParameters.System.Operation.TimeChannels.TC04.OnTime), 
						ADR(SavedInterface.TC.CT4), 
						'UINT', ('Parameters.System.Operation.TimeChannels.TC04.OnTime'), ('CT4'));	
		ExchangeData(	ADR(Parameters.System.Operation.TimeChannels.TC05.OnTime), 
						ADR(ADS_Standard.Tags.Settings.TC.CT5), 
						SIZEOF(Parameters.System.Operation.TimeChannels.TC05.OnTime), 
						ADR(SavedParameters.System.Operation.TimeChannels.TC05.OnTime), 
						ADR(SavedInterface.TC.CT5), 
						'UINT', ('Parameters.System.Operation.TimeChannels.TC05.OnTime'), ('CT5'));	
		ExchangeData(	ADR(Parameters.System.Operation.TimeChannels.TC06.OnTime), 
						ADR(ADS_Standard.Tags.Settings.TC.CT6), 
						SIZEOF(Parameters.System.Operation.TimeChannels.TC06.OnTime), 
						ADR(SavedParameters.System.Operation.TimeChannels.TC06.OnTime), 
						ADR(SavedInterface.TC.CT6), 
						'UINT', ('Parameters.System.Operation.TimeChannels.TC06.OnTime'), ('CT6'));	
		ExchangeData(	ADR(Parameters.System.Operation.TimeChannels.TC07.OnTime), 
						ADR(ADS_Standard.Tags.Settings.TC.CT7), 
						SIZEOF(Parameters.System.Operation.TimeChannels.TC07.OnTime), 
						ADR(SavedParameters.System.Operation.TimeChannels.TC07.OnTime), 
						ADR(SavedInterface.TC.CT7), 
						'UINT', ('Parameters.System.Operation.TimeChannels.TC07.OnTime'), ('CT7'));	

		ExchangeData(	ADR(Parameters.System.Operation.TimeChannels.TC11.OnTime), 
						ADR(ADS_Standard.Tags.Settings.TC.CT11), 
						SIZEOF(Parameters.System.Operation.TimeChannels.TC11.OnTime), 
						ADR(SavedParameters.System.Operation.TimeChannels.TC11.OnTime), 
						ADR(SavedInterface.TC.CT11), 
						'UINT', ('Parameters.System.Operation.TimeChannels.TC11.OnTime'), ('CT11'));	
		ExchangeData(	ADR(Parameters.System.Operation.TimeChannels.TC12.OnTime), 
						ADR(ADS_Standard.Tags.Settings.TC.CT12), 
						SIZEOF(Parameters.System.Operation.TimeChannels.TC12.OnTime), 
						ADR(SavedParameters.System.Operation.TimeChannels.TC12.OnTime), 
						ADR(SavedInterface.TC.CT12), 
						'UINT', ('Parameters.System.Operation.TimeChannels.TC12.OnTime'), ('CT12'));	
		ExchangeData(	ADR(Parameters.System.Operation.TimeChannels.TC13.OnTime), 
						ADR(ADS_Standard.Tags.Settings.TC.CT13), 
						SIZEOF(Parameters.System.Operation.TimeChannels.TC13.OnTime), 
						ADR(SavedParameters.System.Operation.TimeChannels.TC13.OnTime), 
						ADR(SavedInterface.TC.CT13), 
						'UINT', ('Parameters.System.Operation.TimeChannels.TC13.OnTime'), ('CT13'));	
		ExchangeData(	ADR(Parameters.System.Operation.TimeChannels.TC14.OnTime), 
						ADR(ADS_Standard.Tags.Settings.TC.CT14), 
						SIZEOF(Parameters.System.Operation.TimeChannels.TC14.OnTime), 
						ADR(SavedParameters.System.Operation.TimeChannels.TC14.OnTime), 
						ADR(SavedInterface.TC.CT14), 
						'UINT', ('Parameters.System.Operation.TimeChannels.TC14.OnTime'), ('CT14'));	
		ExchangeData(	ADR(Parameters.System.Operation.TimeChannels.TC15.OnTime), 
						ADR(ADS_Standard.Tags.Settings.TC.CT15), 
						SIZEOF(Parameters.System.Operation.TimeChannels.TC15.OnTime), 
						ADR(SavedParameters.System.Operation.TimeChannels.TC15.OnTime), 
						ADR(SavedInterface.TC.CT15), 
						'UINT', ('Parameters.System.Operation.TimeChannels.TC15.OnTime'), ('CT15'));	
		ExchangeData(	ADR(Parameters.System.Operation.TimeChannels.TC16.OnTime), 
						ADR(ADS_Standard.Tags.Settings.TC.CT16), 
						SIZEOF(Parameters.System.Operation.TimeChannels.TC16.OnTime), 
						ADR(SavedParameters.System.Operation.TimeChannels.TC16.OnTime), 
						ADR(SavedInterface.TC.CT16), 
						'UINT', ('Parameters.System.Operation.TimeChannels.TC16.OnTime'), ('CT16'));	
		ExchangeData(	ADR(Parameters.System.Operation.TimeChannels.TC17.OnTime), 
						ADR(ADS_Standard.Tags.Settings.TC.CT17), 
						SIZEOF(Parameters.System.Operation.TimeChannels.TC17.OnTime), 
						ADR(SavedParameters.System.Operation.TimeChannels.TC17.OnTime), 
						ADR(SavedInterface.TC.CT17), 
						'UINT', ('Parameters.System.Operation.TimeChannels.TC17.OnTime'), ('CT17'));	

		ExchangeData(	ADR(Parameters.System.Operation.TimeChannels.TC21.OnTime), 
						ADR(ADS_Standard.Tags.Settings.TC.CT21), 
						SIZEOF(Parameters.System.Operation.TimeChannels.TC21.OnTime), 
						ADR(SavedParameters.System.Operation.TimeChannels.TC21.OnTime), 
						ADR(SavedInterface.TC.CT21), 
						'UINT', ('Parameters.System.Operation.TimeChannels.TC21.OnTime'), ('CT21'));	
		ExchangeData(	ADR(Parameters.System.Operation.TimeChannels.TC22.OnTime), 
						ADR(ADS_Standard.Tags.Settings.TC.CT22), 
						SIZEOF(Parameters.System.Operation.TimeChannels.TC22.OnTime), 
						ADR(SavedParameters.System.Operation.TimeChannels.TC22.OnTime), 
						ADR(SavedInterface.TC.CT22), 
						'UINT', ('Parameters.System.Operation.TimeChannels.TC22.OnTime'), ('CT22'));	
		ExchangeData(	ADR(Parameters.System.Operation.TimeChannels.TC23.OnTime), 
						ADR(ADS_Standard.Tags.Settings.TC.CT23), 
						SIZEOF(Parameters.System.Operation.TimeChannels.TC23.OnTime), 
						ADR(SavedParameters.System.Operation.TimeChannels.TC23.OnTime), 
						ADR(SavedInterface.TC.CT23), 
						'UINT', ('Parameters.System.Operation.TimeChannels.TC23.OnTime'), ('CT23'));	
		ExchangeData(	ADR(Parameters.System.Operation.TimeChannels.TC24.OnTime), 
						ADR(ADS_Standard.Tags.Settings.TC.CT24), 
						SIZEOF(Parameters.System.Operation.TimeChannels.TC24.OnTime), 
						ADR(SavedParameters.System.Operation.TimeChannels.TC24.OnTime), 
						ADR(SavedInterface.TC.CT24), 
						'UINT', ('Parameters.System.Operation.TimeChannels.TC24.OnTime'), ('CT24'));	
		ExchangeData(	ADR(Parameters.System.Operation.TimeChannels.TC25.OnTime), 
						ADR(ADS_Standard.Tags.Settings.TC.CT25), 
						SIZEOF(Parameters.System.Operation.TimeChannels.TC25.OnTime), 
						ADR(SavedParameters.System.Operation.TimeChannels.TC25.OnTime), 
						ADR(SavedInterface.TC.CT25), 
						'UINT', ('Parameters.System.Operation.TimeChannels.TC25.OnTime'), ('CT25'));	
		ExchangeData(	ADR(Parameters.System.Operation.TimeChannels.TC26.OnTime), 
						ADR(ADS_Standard.Tags.Settings.TC.CT26), 
						SIZEOF(Parameters.System.Operation.TimeChannels.TC26.OnTime), 
						ADR(SavedParameters.System.Operation.TimeChannels.TC26.OnTime), 
						ADR(SavedInterface.TC.CT26), 
						'UINT', ('Parameters.System.Operation.TimeChannels.TC26.OnTime'), ('CT26'));	
		ExchangeData(	ADR(Parameters.System.Operation.TimeChannels.TC27.OnTime), 
						ADR(ADS_Standard.Tags.Settings.TC.CT27), 
						SIZEOF(Parameters.System.Operation.TimeChannels.TC27.OnTime), 
						ADR(SavedParameters.System.Operation.TimeChannels.TC27.OnTime), 
						ADR(SavedInterface.TC.CT27), 
						'UINT', ('Parameters.System.Operation.TimeChannels.TC27.OnTime'), ('CT27'));	

		ExchangeData(	ADR(Parameters.Regulation.SupplyAir.ControlMode), 
						ADR(ADS_Standard.Tags.Settings.SupplyFanControlMode), 
						SIZEOF(Parameters.Regulation.SupplyAir.ControlMode), 
						ADR(SavedParameters.Regulation.Temperature.TemperatureControlSource), 
						ADR(SavedInterface.SupplyFanControlMode), 
						'INT', ('Parameters.Regulation.SupplyAir.ControlMode'), ('SupplyFanControlMode'));	
		
		ExchangeData_LREAL_REAL(	ADR(Parameters.Regulation.SupplyAir.Control.SP), 
						ADR(ADS_Standard.Tags.Settings.SupplyFan_SP), 
						ADR(SavedParameters.Regulation.SupplyAir.Control.SP), 
						ADR(SavedInterface.SupplyFan_SP), 
						('Parameters.Regulation.SupplyAir.Control.SP'), ('SupplyFan_SP'));	
		
		ExchangeData_LREAL_REAL(	ADR(Parameters.Regulation.SupplyAir.Control.SP_HighSpeed), 
						ADR(ADS_Standard.Tags.Settings.SupplyFanHighSpeed_SP), 
						ADR(SavedParameters.Regulation.SupplyAir.Control.SP_HighSpeed), 
						ADR(SavedInterface.SupplyFanHighSpeed_SP), 
						('Parameters.Regulation.SupplyAir.Control.SP_HighSpeed'), ('SupplyFanHighSpeed_SP'));	
		
		ExchangeData_LREAL_REAL(	ADR(Parameters.Regulation.SupplyAir.Control.P), 
						ADR(ADS_Standard.Tags.Settings.SupplyFanControl_P), 
						ADR(SavedParameters.Regulation.SupplyAir.Control.P), 
						ADR(SavedInterface.SupplyFanControl_P), 
						('Parameters.Regulation.SupplyAir.Control.P'), ('SupplyFanControl_P'));	
		
		ExchangeData(	ADR(Parameters.Regulation.SupplyAir.Control.I), 
						ADR(ADS_Standard.Tags.Settings.SupplyFanControl_I), 
						SIZEOF(Parameters.Regulation.SupplyAir.Control.I),
						ADR(SavedParameters.Regulation.SupplyAir.Control.I), 
						ADR(SavedInterface.SupplyFanControl_I), 
						'TIME', ('Parameters.Regulation.SupplyAir.Control.I'), ('SupplyFanControl_I'));	
		
		ExchangeData(	ADR(Parameters.Regulation.SupplyAir.SetPointAdjustment.Curve), 
						ADR(ADS_Standard.Tags.Settings.T_GQ1_CURVE), 
						SIZEOF(Parameters.Regulation.SupplyAir.SetPointAdjustment.Curve), 
						ADR(SavedParameters.Regulation.SupplyAir.SetPointAdjustment.Curve), 
						ADR(SavedInterface.T_GQ1_CURVE), 
						'SetPointOffsetCurve', ('Parameters.Regulation.SupplyAir.SetPointAdjustment.Curve'), ('T_GQ1_CURVE'));	
		
